LIN {X 0,Y 325.669,Z 599.39,A -85,B 0,C 180,E1 -14857.439,E2 -14857.439} C_VEL
LIN {X 0,Y 325.677,Z 594.579,A -85,B 0,C 180,E1 -14859.314,E2 -14859.314} C_VEL
LIN {X 0,Y 326.028,Z 587.351,A -85,B 0,C 180,E1 -14861.501,E2 -14861.501} C_VEL
LIN {X 0,Y 326.643,Z 579.568,A -85,B 0,C 180,E1 -14863.373,E2 -14863.373} C_VEL
LIN {X 0,Y 327.397,Z 571.651,A -85,B 0,C 180,E1 -14864.927,E2 -14864.927} C_VEL
LIN {X 0,Y 328.601,Z 562.062,A -85,B 0,C 180,E1 -14866.462,E2 -14866.462} C_VEL
LIN {X 0,Y 329.683,Z 551.406,A -85,B 0,C 180,E1 -14867.845,E2 -14867.845} C_VEL
LIN {X 0,Y 329.651,Z 539.37,A -85,B 0,C 180,E1 -14869.134,E2 -14869.134} C_VEL
LIN {X 0,Y 329.259,Z 526.597,A -85,B 0,C 180,E1 -14870.206,E2 -14870.206} C_VEL
LIN {X 0,Y 328.339,Z 513.613,A -85,B 0,C 180,E1 -14871.05,E2 -14871.05} C_VEL
LIN {X 0,Y 326.76,Z 500.315,A -85,B 0,C 180,E1 -14871.695,E2 -14871.695} C_VEL
LIN {X 0,Y 326.159,Z 495.999,A -85,B 0,C 180,E1 -14871.874,E2 -14871.874} C_VEL
LIN {X 0,Y 327.015,Z 484.007,A -85,B 0,C 180,E1 -14876.14,E2 -14876.14} C_VEL
LIN {X 0,Y 328.094,Z 472.597,A -85,B 0,C 180,E1 -14880.224,E2 -14880.224} C_VEL
LIN {X 0,Y 329.193,Z 462.925,A -85,B 0,C 180,E1 -14883.716,E2 -14883.716} C_VEL
LIN {X 0,Y 330.448,Z 453.169,A -85,B 0,C 180,E1 -14887.311,E2 -14887.311} C_VEL
LIN {X 0,Y 330.5,Z 451.076,A -85,B 0,C 180,E1 -14888.113,E2 -14888.113} C_VEL
LIN {X 0,Y 328.983,Z 442.588,A -85,B 0,C 180,E1 -14891.609,E2 -14891.609} C_VEL
LIN {X 0,Y 327.405,Z 434.615,A -85,B 0,C 180,E1 -14895.102,E2 -14895.102} C_VEL
LIN {X 0,Y 326.602,Z 430.809,A -85,B 0,C 180,E1 -14896.887,E2 -14896.887} C_VEL
LIN {X 0,Y 326.612,Z 430.8,A -85,B 0,C 180,E1 -14900.772,E2 -14900.772} C_VEL
LIN {X 0,Y 326.614,Z 430.802,A -85,B 0,C 180,E1 -14904.481,E2 -14904.481} C_VEL
LIN {X 0,Y 326.61,Z 430.799,A -85,B 0,C 180,E1 -14907.456,E2 -14907.456} C_VEL
LIN {X 0,Y 326.648,Z 430.798,A -85,B 0,C 180,E1 -14910.34,E2 -14910.34} C_VEL
LIN {X 0,Y 326.69,Z 430.791,A -85,B 0,C 180,E1 -14914.516,E2 -14914.516} C_VEL
LIN {X 0,Y 326.649,Z 430.796,A -85,B 0,C 180,E1 -14918.546,E2 -14918.546} C_VEL
LIN {X 0,Y 326.745,Z 430.782,A -85,B 0,C 180,E1 -14921.178,E2 -14921.178} C_VEL
LIN {X 0,Y 326.764,Z 430.78,A -85,B 0,C 180,E1 -14925.433,E2 -14925.433} C_VEL
LIN {X 0,Y 326.774,Z 430.778,A -85,B 0,C 180,E1 -14928.839,E2 -14928.839} C_VEL
LIN {X 0,Y 326.945,Z 430.758,A -85,B 0,C 180,E1 -14932.59,E2 -14932.59} C_VEL
LIN {X 0,Y 326.986,Z 430.755,A -85,B 0,C 180,E1 -14933.831,E2 -14933.831} C_VEL
LIN {X 0,Y 327.05,Z 430.745,A -85,B 0,C 180,E1 -14937.537,E2 -14937.537} C_VEL
LIN {X 0,Y 327.218,Z 430.728,A -85,B 0,C 180,E1 -14940,E2 -14940} C_VEL
LIN {X 0,Y 327.047,Z 430.745,A -85,B 0,C 180,E1 -14942.463,E2 -14942.463} C_VEL
LIN {X 0,Y 326.972,Z 430.752,A -85,B 0,C 180,E1 -14946.678,E2 -14946.678} C_VEL
LIN {X 0,Y 326.815,Z 430.777,A -85,B 0,C 180,E1 -14949.906,E2 -14949.906} C_VEL
LIN {X 0,Y 326.76,Z 430.78,A -85,B 0,C 180,E1 -14953.686,E2 -14953.686} C_VEL
LIN {X 0,Y 326.701,Z 430.788,A -85,B 0,C 180,E1 -14957.528,E2 -14957.528} C_VEL
LIN {X 0,Y 326.666,Z 430.79,A -85,B 0,C 180,E1 -14960.135,E2 -14960.135} C_VEL
LIN {X 0,Y 326.653,Z 430.794,A -85,B 0,C 180,E1 -14964.129,E2 -14964.129} C_VEL
LIN {X 0,Y 326.684,Z 430.788,A -85,B 0,C 180,E1 -14966.858,E2 -14966.858} C_VEL
LIN {X 0,Y 326.635,Z 430.794,A -85,B 0,C 180,E1 -14970.61,E2 -14970.61} C_VEL
LIN {X 0,Y 326.609,Z 430.8,A -85,B 0,C 180,E1 -14974.02,E2 -14974.02} C_VEL
LIN {X 0,Y 326.629,Z 430.796,A -85,B 0,C 180,E1 -14977.239,E2 -14977.239} C_VEL
LIN {X 0,Y 326.579,Z 430.801,A -85,B 0,C 180,E1 -14981.132,E2 -14981.132} C_VEL
LIN {X 0,Y 326.53,Z 430.807,A -85,B 0,C 180,E1 -14984.743,E2 -14984.743} C_VEL
LIN {X 0,Y 326.578,Z 430.803,A -85,B 0,C 180,E1 -14988.155,E2 -14988.155} C_VEL
LIN {X 0,Y 326.626,Z 430.797,A -85,B 0,C 180,E1 -14991.392,E2 -14991.392} C_VEL
LIN {X 0,Y 326.622,Z 430.795,A -85,B 0,C 180,E1 -14994.852,E2 -14994.852} C_VEL
LIN {X 0,Y 326.618,Z 430.799,A -85,B 0,C 180,E1 -14997.457,E2 -14997.457} C_VEL
LIN {X 0,Y 326.664,Z 430.79,A -85,B 0,C 180,E1 -15000.342,E2 -15000.342} C_VEL
LIN {X 0,Y 326.688,Z 430.789,A -85,B 0,C 180,E1 -15003.143,E2 -15003.143} C_VEL
LIN {X 0,Y 326.655,Z 430.797,A -85,B 0,C 180,E1 -15005.872,E2 -15005.872} C_VEL
LIN {X 0,Y 326.671,Z 430.795,A -85,B 0,C 180,E1 -15009.866,E2 -15009.866} C_VEL
LIN {X 0,Y 326.767,Z 430.78,A -85,B 0,C 180,E1 -15012.234,E2 -15012.234} C_VEL
LIN {X 0,Y 330.786,Z 443.096,A -85,B 0,C 180,E1 -15013.451,E2 -15013.451} C_VEL
LIN {X 0,Y 333.898,Z 454.069,A -85,B 0,C 180,E1 -15014.746,E2 -15014.746} C_VEL
LIN {X 0,Y 333.148,Z 464.325,A -85,B 0,C 180,E1 -15015.961,E2 -15015.961} C_VEL
LIN {X 0,Y 331.99,Z 474.107,A -85,B 0,C 180,E1 -15017.371,E2 -15017.371} C_VEL
LIN {X 0,Y 330.794,Z 483.132,A -85,B 0,C 180,E1 -15018.977,E2 -15018.977} C_VEL
LIN {X 0,Y 329.724,Z 491.285,A -85,B 0,C 180,E1 -15020.801,E2 -15020.801} C_VEL
LIN {X 0,Y 328.764,Z 497.856,A -85,B 0,C 180,E1 -15022.631,E2 -15022.631} C_VEL
LIN {X 0,Y 328.229,Z 503.065,A -85,B 0,C 180,E1 -15024.471,E2 -15024.471} C_VEL
LIN {X 0,Y 327.548,Z 507.179,A -85,B 0,C 180,E1 -15026.31,E2 -15026.31} C_VEL
LIN {X 0,Y 327.213,Z 509.362,A -85,B 0,C 180,E1 -15027.538,E2 -15027.538} C_VEL
LIN {X 0,Y 326.991,Z 511.075,A -85,B 0,C 180,E1 -15028.769,E2 -15028.769} C_VEL
LIN {X 0,Y 326.874,Z 513.281,A -85,B 0,C 180,E1 -15031.232,E2 -15031.232} C_VEL
LIN {X 0,Y 326.764,Z 513.841,A -85,B 0,C 180,E1 -15032.466,E2 -15032.466} C_VEL
LIN {X 0,Y 326.652,Z 513.995,A -85,B 0,C 180,E1 -15033.701,E2 -15033.701} C_VEL
LIN {X 0,Y 327.059,Z 513.1,A -85,B 0,C 180,E1 -15036.168,E2 -15036.168} C_VEL
LIN {X 0,Y 327.451,Z 512.077,A -85,B 0,C 180,E1 -15037.399,E2 -15037.399} C_VEL
LIN {X 0,Y 328.031,Z 508.988,A -85,B 0,C 180,E1 -15039.752,E2 -15039.752} C_VEL
LIN {X 0,Y 328.83,Z 505.182,A -85,B 0,C 180,E1 -15041.715,E2 -15041.715} C_VEL
LIN {X 0,Y 329.619,Z 500.482,A -85,B 0,C 180,E1 -15043.565,E2 -15043.565} C_VEL
LIN {X 0,Y 330.597,Z 494.526,A -85,B 0,C 180,E1 -15045.411,E2 -15045.411} C_VEL
LIN {X 0,Y 331.772,Z 487.085,A -85,B 0,C 180,E1 -15047.252,E2 -15047.252} C_VEL
LIN {X 0,Y 333.026,Z 479.414,A -85,B 0,C 180,E1 -15048.774,E2 -15048.774} C_VEL
LIN {X 0,Y 334.289,Z 468.983,A -85,B 0,C 180,E1 -15050.458,E2 -15050.458} C_VEL
LIN {X 0,Y 335.431,Z 459.35,A -85,B 0,C 180,E1 -15051.7,E2 -15051.7} C_VEL
LIN {X 0,Y 335.445,Z 457.058,A -85,B 0,C 180,E1 -15051.978,E2 -15051.978} C_VEL
LIN {X 0,Y 332.16,Z 446.15,A -85,B 0,C 180,E1 -15053.401,E2 -15053.401} C_VEL
LIN {X 0,Y 328.166,Z 435.083,A -85,B 0,C 180,E1 -15054.651,E2 -15054.651} C_VEL
LIN {X 0,Y 326.687,Z 430.788,A -85,B 0,C 180,E1 -15055.101,E2 -15055.101} C_VEL
LIN {X 0,Y 326.66,Z 430.797,A -85,B 0,C 180,E1 -15058.251,E2 -15058.251} C_VEL
LIN {X 0,Y 326.598,Z 430.801,A -85,B 0,C 180,E1 -15061.095,E2 -15061.095} C_VEL
LIN {X 0,Y 326.612,Z 430.803,A -85,B 0,C 180,E1 -15064.019,E2 -15064.019} C_VEL
LIN {X 0,Y 326.631,Z 430.796,A -85,B 0,C 180,E1 -15067.239,E2 -15067.239} C_VEL
LIN {X 0,Y 326.581,Z 430.802,A -85,B 0,C 180,E1 -15071.131,E2 -15071.131} C_VEL
LIN {X 0,Y 326.532,Z 430.808,A -85,B 0,C 180,E1 -15074.743,E2 -15074.743} C_VEL
LIN {X 0,Y 326.58,Z 430.806,A -85,B 0,C 180,E1 -15078.154,E2 -15078.154} C_VEL
LIN {X 0,Y 326.627,Z 430.796,A -85,B 0,C 180,E1 -15081.391,E2 -15081.391} C_VEL
LIN {X 0,Y 326.623,Z 430.796,A -85,B 0,C 180,E1 -15084.851,E2 -15084.851} C_VEL
LIN {X 0,Y 326.614,Z 430.799,A -85,B 0,C 180,E1 -15087.456,E2 -15087.456} C_VEL
LIN {X 0,Y 326.664,Z 430.793,A -85,B 0,C 180,E1 -15090.341,E2 -15090.341} C_VEL
LIN {X 0,Y 326.694,Z 430.788,A -85,B 0,C 180,E1 -15094.516,E2 -15094.516} C_VEL
LIN {X 0,Y 326.655,Z 430.792,A -85,B 0,C 180,E1 -15095.197,E2 -15095.197} C_VEL
LIN {X 0,Y 325.957,Z 430.883,A -85,B 0,C 180,E1 -15096.225,E2 -15096.225} C_VEL
LIN {X 0,Y 323.068,Z 431.244,A -85,B 0,C 180,E1 -15097.898,E2 -15097.898} C_VEL
LIN {X 0,Y 320.677,Z 431.538,A -85,B 0,C 180,E1 -15099.254,E2 -15099.254} C_VEL
LIN {X 0,Y 319.714,Z 431.658,A -85,B 0,C 180,E1 -15100.304,E2 -15100.304} C_VEL
LIN {X 0,Y 319.668,Z 431.662,A -85,B 0,C 180,E1 -15100.659,E2 -15100.659} C_VEL
LIN {X 0,Y 319.742,Z 431.745,A -85,B 0,C 180,E1 -15102.367,E2 -15102.367} C_VEL
LIN {X 0,Y 322.789,Z 444.313,A -85,B 0,C 180,E1 -15103.558,E2 -15103.558} C_VEL
LIN {X 0,Y 323.928,Z 449.817,A -85,B 0,C 180,E1 -15104.161,E2 -15104.161} C_VEL
LIN {X 0,Y 323.077,Z 461.417,A -85,B 0,C 180,E1 -15105.513,E2 -15105.513} C_VEL
LIN {X 0,Y 322.358,Z 472.344,A -85,B 0,C 180,E1 -15107.087,E2 -15107.087} C_VEL
LIN {X 0,Y 321.437,Z 483.009,A -85,B 0,C 180,E1 -15108.97,E2 -15108.97} C_VEL
LIN {X 0,Y 320.873,Z 491.396,A -85,B 0,C 180,E1 -15110.814,E2 -15110.814} C_VEL
LIN {X 0,Y 320.306,Z 498.633,A -85,B 0,C 180,E1 -15112.752,E2 -15112.752} C_VEL
LIN {X 0,Y 319.786,Z 505.159,A -85,B 0,C 180,E1 -15114.956,E2 -15114.956} C_VEL
LIN {X 0,Y 319.604,Z 509.482,A -85,B 0,C 180,E1 -15116.848,E2 -15116.848} C_VEL
LIN {X 0,Y 319.665,Z 512.75,A -85,B 0,C 180,E1 -15118.74,E2 -15118.74} C_VEL
LIN {X 0,Y 319.823,Z 514.387,A -85,B 0,C 180,E1 -15120,E2 -15120} C_VEL
LIN {X 0,Y 319.913,Z 515.65,A -85,B 0,C 180,E1 -15121.259,E2 -15121.259} C_VEL
LIN {X 0,Y 320.345,Z 516.87,A -85,B 0,C 180,E1 -15123.774,E2 -15123.774} C_VEL
LIN {X 0,Y 320.674,Z 516.901,A -85,B 0,C 180,E1 -15125.029,E2 -15125.029} C_VEL
LIN {X 0,Y 321.105,Z 516.495,A -85,B 0,C 180,E1 -15126.283,E2 -15126.283} C_VEL
LIN {X 0,Y 322.298,Z 514.492,A -85,B 0,C 180,E1 -15128.78,E2 -15128.78} C_VEL
LIN {X 0,Y 323.367,Z 511.902,A -85,B 0,C 180,E1 -15130.646,E2 -15130.646} C_VEL
LIN {X 0,Y 324.733,Z 508.273,A -85,B 0,C 180,E1 -15132.499,E2 -15132.499} C_VEL
LIN {X 0,Y 326.445,Z 502.775,A -85,B 0,C 180,E1 -15134.621,E2 -15134.621} C_VEL
LIN {X 0,Y 328.227,Z 496.576,A -85,B 0,C 180,E1 -15136.482,E2 -15136.482} C_VEL
LIN {X 0,Y 330.281,Z 488.982,A -85,B 0,C 180,E1 -15138.292,E2 -15138.292} C_VEL
LIN {X 0,Y 332.466,Z 479.622,A -85,B 0,C 180,E1 -15140.091,E2 -15140.091} C_VEL
LIN {X 0,Y 334.516,Z 470.377,A -85,B 0,C 180,E1 -15141.521,E2 -15141.521} C_VEL
LIN {X 0,Y 335.117,Z 467.023,A -85,B 0,C 180,E1 -15141.982,E2 -15141.982} C_VEL
LIN {X 0,Y 332.872,Z 458.578,A -85,B 0,C 180,E1 -15143.65,E2 -15143.65} C_VEL
LIN {X 0,Y 329.131,Z 449.041,A -85,B 0,C 180,E1 -15145.596,E2 -15145.596} C_VEL
LIN {X 0,Y 324.805,Z 440.543,A -85,B 0,C 180,E1 -15147.483,E2 -15147.483} C_VEL
LIN {X 0,Y 322.807,Z 437.235,A -85,B 0,C 180,E1 -15148.282,E2 -15148.282} C_VEL
LIN {X 0,Y 320.236,Z 433.853,A -85,B 0,C 180,E1 -15149.259,E2 -15149.259} C_VEL
LIN {X 0,Y 319.626,Z 431.669,A -85,B 0,C 180,E1 -15149.652,E2 -15149.652} C_VEL
LIN {X 0,Y 319.579,Z 431.674,A -85,B 0,C 180,E1 -15153.352,E2 -15153.352} C_VEL
LIN {X 0,Y 319.561,Z 431.681,A -85,B 0,C 180,E1 -15156.427,E2 -15156.427} C_VEL
LIN {X 0,Y 319.565,Z 431.681,A -85,B 0,C 180,E1 -15160.449,E2 -15160.449} C_VEL
LIN {X 0,Y 319.588,Z 431.813,A -85,B 0,C 180,E1 -15160.861,E2 -15160.861} C_VEL
LIN {X 0,Y 321.083,Z 439.049,A -85,B 0,C 180,E1 -15164.461,E2 -15164.461} C_VEL
LIN {X 0,Y 322.551,Z 446.207,A -85,B 0,C 180,E1 -15167.801,E2 -15167.801} C_VEL
LIN {X 0,Y 323.926,Z 453.523,A -85,B 0,C 180,E1 -15171.009,E2 -15171.009} C_VEL
LIN {X 0,Y 324.151,Z 455.88,A -85,B 0,C 180,E1 -15171.991,E2 -15171.991} C_VEL
LIN {X 0,Y 322.624,Z 465.941,A -85,B 0,C 180,E1 -15175.872,E2 -15175.872} C_VEL
LIN {X 0,Y 321.265,Z 476.33,A -85,B 0,C 180,E1 -15179.791,E2 -15179.791} C_VEL
LIN {X 0,Y 320.595,Z 482.587,A -85,B 0,C 180,E1 -15182.058,E2 -15182.058} C_VEL
LIN {X 0,Y 321.374,Z 486.979,A -85,B 0,C 180,E1 -15182.529,E2 -15182.529} C_VEL
LIN {X 0,Y 323.338,Z 495.524,A -85,B 0,C 180,E1 -15183.548,E2 -15183.548} C_VEL
LIN {X 0,Y 325.59,Z 511.177,A -85,B 0,C 180,E1 -15185.304,E2 -15185.304} C_VEL
LIN {X 0,Y 326.507,Z 524.117,A -85,B 0,C 180,E1 -15186.797,E2 -15186.797} C_VEL
LIN {X 0,Y 326.004,Z 535.939,A -85,B 0,C 180,E1 -15188.199,E2 -15188.199} C_VEL
LIN {X 0,Y 324.904,Z 548.75,A -85,B 0,C 180,E1 -15189.916,E2 -15189.916} C_VEL
LIN {X 0,Y 323.91,Z 557.8,A -85,B 0,C 180,E1 -15191.334,E2 -15191.334} C_VEL
LIN {X 0,Y 321.843,Z 568.154,A -85,B 0,C 180,E1 -15193.181,E2 -15193.181} C_VEL
LIN {X 0,Y 319.919,Z 581.019,A -85,B 0,C 180,E1 -15196.016,E2 -15196.016} C_VEL
LIN {X 0,Y 319.057,Z 588.233,A -85,B 0,C 180,E1 -15197.921,E2 -15197.921} C_VEL
LIN {X 0,Y 318.563,Z 594.058,A -85,B 0,C 180,E1 -15199.834,E2 -15199.834} C_VEL
LIN {X 0,Y 318.512,Z 598.707,A -85,B 0,C 180,E1 -15201.754,E2 -15201.754} C_VEL
LIN {X 0,Y 318.634,Z 602.266,A -85,B 0,C 180,E1 -15203.668,E2 -15203.668} C_VEL
LIN {X 0,Y 318.818,Z 604.062,A -85,B 0,C 180,E1 -15204.941,E2 -15204.941} C_VEL
LIN {X 0,Y 318.996,Z 605.438,A -85,B 0,C 180,E1 -15206.21,E2 -15206.21} C_VEL
LIN {X 0,Y 319.08,Z 606.386,A -85,B 0,C 180,E1 -15207.475,E2 -15207.475} C_VEL
LIN {X 0,Y 319.469,Z 606.925,A -85,B 0,C 180,E1 -15208.739,E2 -15208.739} C_VEL
LIN {X 0,Y 319.619,Z 607.015,A -85,B 0,C 180,E1 -15210,E2 -15210} C_VEL
LIN {X 0,Y 319.487,Z 606.66,A -85,B 0,C 180,E1 -15211.26,E2 -15211.26} C_VEL
LIN {X 0,Y 319.132,Z 605.866,A -85,B 0,C 180,E1 -15212.524,E2 -15212.524} C_VEL
LIN {X 0,Y 319.046,Z 604.651,A -85,B 0,C 180,E1 -15213.789,E2 -15213.789} C_VEL
LIN {X 0,Y 318.806,Z 602.006,A -85,B 0,C 180,E1 -15215.693,E2 -15215.693} C_VEL
LIN {X 0,Y 318.604,Z 598.302,A -85,B 0,C 180,E1 -15217.605,E2 -15217.605} C_VEL
LIN {X 0,Y 318.615,Z 593.468,A -85,B 0,C 180,E1 -15219.522,E2 -15219.522} C_VEL
LIN {X 0,Y 319.018,Z 586.22,A -85,B 0,C 180,E1 -15221.758,E2 -15221.758} C_VEL
LIN {X 0,Y 319.692,Z 578.418,A -85,B 0,C 180,E1 -15223.669,E2 -15223.669} C_VEL
LIN {X 0,Y 320.297,Z 571.806,A -85,B 0,C 180,E1 -15225.005,E2 -15225.005} C_VEL
LIN {X 0,Y 321.504,Z 562.93,A -85,B 0,C 180,E1 -15226.509,E2 -15226.509} C_VEL
LIN {X 0,Y 322.676,Z 552.778,A -85,B 0,C 180,E1 -15227.917,E2 -15227.917} C_VEL
LIN {X 0,Y 322.689,Z 541.461,A -85,B 0,C 180,E1 -15229.215,E2 -15229.215} C_VEL
LIN {X 0,Y 322.447,Z 528.376,A -85,B 0,C 180,E1 -15230.41,E2 -15230.41} C_VEL
LIN {X 0,Y 321.673,Z 515.529,A -85,B 0,C 180,E1 -15231.319,E2 -15231.319} C_VEL
LIN {X 0,Y 320.175,Z 502.104,A -85,B 0,C 180,E1 -15232.032,E2 -15232.032} C_VEL
LIN {X 0,Y 319.167,Z 494.914,A -85,B 0,C 180,E1 -15232.357,E2 -15232.357} C_VEL
LIN {X 0,Y 320.089,Z 482.916,A -85,B 0,C 180,E1 -15236.75,E2 -15236.75} C_VEL
LIN {X 0,Y 321.44,Z 470.016,A -85,B 0,C 180,E1 -15241.493,E2 -15241.493} C_VEL
LIN {X 0,Y 322.624,Z 459.929,A -85,B 0,C 180,E1 -15245.259,E2 -15245.259} C_VEL
LIN {X 0,Y 323.456,Z 454.085,A -85,B 0,C 180,E1 -15247.472,E2 -15247.472} C_VEL
LIN {X 0,Y 323.155,Z 450.05,A -85,B 0,C 180,E1 -15249.101,E2 -15249.101} C_VEL
LIN {X 0,Y 321.624,Z 441.786,A -85,B 0,C 180,E1 -15252.641,E2 -15252.641} C_VEL
LIN {X 0,Y 319.907,Z 433.467,A -85,B 0,C 180,E1 -15256.466,E2 -15256.466} C_VEL
LIN {X 0,Y 319.535,Z 431.689,A -85,B 0,C 180,E1 -15257.39,E2 -15257.39} C_VEL
LIN {X 0,Y 319.548,Z 431.683,A -85,B 0,C 180,E1 -15260.371,E2 -15260.371} C_VEL
LIN {X 0,Y 319.56,Z 431.678,A -85,B 0,C 180,E1 -15263.573,E2 -15263.573} C_VEL
LIN {X 0,Y 319.577,Z 431.677,A -85,B 0,C 180,E1 -15266.686,E2 -15266.686} C_VEL
LIN {X 0,Y 319.585,Z 431.675,A -85,B 0,C 180,E1 -15269.616,E2 -15269.616} C_VEL
LIN {X 0,Y 319.606,Z 431.673,A -85,B 0,C 180,E1 -15272.498,E2 -15272.498} C_VEL
LIN {X 0,Y 319.605,Z 431.671,A -85,B 0,C 180,E1 -15275.304,E2 -15275.304} C_VEL
LIN {X 0,Y 319.598,Z 431.677,A -85,B 0,C 180,E1 -15278.048,E2 -15278.048} C_VEL
LIN {X 0,Y 319.69,Z 431.661,A -85,B 0,C 180,E1 -15280.962,E2 -15280.962} C_VEL
LIN {X 0,Y 319.731,Z 431.656,A -85,B 0,C 180,E1 -15285.276,E2 -15285.276} C_VEL
LIN {X 0,Y 319.754,Z 431.656,A -85,B 0,C 180,E1 -15289.873,E2 -15289.873} C_VEL
LIN {X 0,Y 319.939,Z 431.631,A -85,B 0,C 180,E1 -15293.694,E2 -15293.694} C_VEL
LIN {X 0,Y 319.994,Z 431.623,A -85,B 0,C 180,E1 -15297.483,E2 -15297.483} C_VEL
LIN {X 0,Y 320.17,Z 431.606,A -85,B 0,C 180,E1 -15300,E2 -15300} C_VEL
LIN {X 0,Y 319.991,Z 431.624,A -85,B 0,C 180,E1 -15302.518,E2 -15302.518} C_VEL
LIN {X 0,Y 319.932,Z 431.629,A -85,B 0,C 180,E1 -15306.669,E2 -15306.669} C_VEL
LIN {X 0,Y 319.759,Z 431.655,A -85,B 0,C 180,E1 -15310.127,E2 -15310.127} C_VEL
LIN {X 0,Y 319.732,Z 431.654,A -85,B 0,C 180,E1 -15314.725,E2 -15314.725} C_VEL
LIN {X 0,Y 319.69,Z 431.658,A -85,B 0,C 180,E1 -15319.038,E2 -15319.038} C_VEL
LIN {X 0,Y 319.571,Z 431.669,A -85,B 0,C 180,E1 -15323.32,E2 -15323.32} C_VEL
LIN {X 0,Y 319.635,Z 431.67,A -85,B 0,C 180,E1 -15326.088,E2 -15326.088} C_VEL
LIN {X 0,Y 319.581,Z 431.673,A -85,B 0,C 180,E1 -15328.935,E2 -15328.935} C_VEL
LIN {X 0,Y 319.533,Z 431.68,A -85,B 0,C 180,E1 -15331.862,E2 -15331.862} C_VEL
LIN {X 0,Y 319.581,Z 431.673,A -85,B 0,C 180,E1 -15335.543,E2 -15335.543} C_VEL
LIN {X 0,Y 319.575,Z 431.678,A -85,B 0,C 180,E1 -15338.008,E2 -15338.008} C_VEL
LIN {X 0,Y 319.527,Z 431.683,A -85,B 0,C 180,E1 -15341.597,E2 -15341.597} C_VEL
LIN {X 0,Y 319.491,Z 431.684,A -85,B 0,C 180,E1 -15345.258,E2 -15345.258} C_VEL
LIN {X 0,Y 319.53,Z 431.678,A -85,B 0,C 180,E1 -15348.712,E2 -15348.712} C_VEL
LIN {X 0,Y 319.579,Z 431.674,A -85,B 0,C 180,E1 -15352.344,E2 -15352.344} C_VEL
LIN {X 0,Y 319.563,Z 431.675,A -85,B 0,C 180,E1 -15355.124,E2 -15355.124} C_VEL
LIN {X 0,Y 319.577,Z 431.674,A -85,B 0,C 180,E1 -15359.057,E2 -15359.057} C_VEL
LIN {X 0,Y 319.62,Z 431.669,A -85,B 0,C 180,E1 -15362.499,E2 -15362.499} C_VEL
LIN {X 0,Y 319.608,Z 431.672,A -85,B 0,C 180,E1 -15365.304,E2 -15365.304} C_VEL
LIN {X 0,Y 319.601,Z 431.675,A -85,B 0,C 180,E1 -15368.048,E2 -15368.048} C_VEL
LIN {X 0,Y 319.744,Z 431.655,A -85,B 0,C 180,E1 -15371.782,E2 -15371.782} C_VEL
LIN {X 0,Y 323.953,Z 444.512,A -85,B 0,C 180,E1 -15373.084,E2 -15373.084} C_VEL
LIN {X 0,Y 327.063,Z 455.441,A -85,B 0,C 180,E1 -15374.419,E2 -15374.419} C_VEL
LIN {X 0,Y 326.814,Z 460.778,A -85,B 0,C 180,E1 -15375.046,E2 -15375.046} C_VEL
LIN {X 0,Y 325.617,Z 471.249,A -85,B 0,C 180,E1 -15376.451,E2 -15376.451} C_VEL
LIN {X 0,Y 324.617,Z 479.482,A -85,B 0,C 180,E1 -15377.814,E2 -15377.814} C_VEL
LIN {X 0,Y 323.586,Z 487.223,A -85,B 0,C 180,E1 -15379.362,E2 -15379.362} C_VEL
LIN {X 0,Y 322.425,Z 494.811,A -85,B 0,C 180,E1 -15381.224,E2 -15381.224} C_VEL
LIN {X 0,Y 321.694,Z 500.842,A -85,B 0,C 180,E1 -15383.099,E2 -15383.099} C_VEL
LIN {X 0,Y 320.985,Z 505.658,A -85,B 0,C 180,E1 -15384.976,E2 -15384.976} C_VEL
LIN {X 0,Y 320.398,Z 509.39,A -85,B 0,C 180,E1 -15386.857,E2 -15386.857} C_VEL
LIN {X 0,Y 319.97,Z 512.13,A -85,B 0,C 180,E1 -15388.742,E2 -15388.742} C_VEL
LIN {X 0,Y 319.852,Z 514.316,A -85,B 0,C 180,E1 -15391.259,E2 -15391.259} C_VEL
LIN {X 0,Y 319.74,Z 514.865,A -85,B 0,C 180,E1 -15392.52,E2 -15392.52} C_VEL
LIN {X 0,Y 319.631,Z 515.003,A -85,B 0,C 180,E1 -15393.782,E2 -15393.782} C_VEL
LIN {X 0,Y 320.067,Z 514.088,A -85,B 0,C 180,E1 -15396.303,E2 -15396.303} C_VEL
LIN {X 0,Y 320.477,Z 513.053,A -85,B 0,C 180,E1 -15397.561,E2 -15397.561} C_VEL
LIN {X 0,Y 321.106,Z 509.937,A -85,B 0,C 180,E1 -15399.964,E2 -15399.964} C_VEL
LIN {X 0,Y 321.946,Z 506.107,A -85,B 0,C 180,E1 -15401.969,E2 -15401.969} C_VEL
LIN {X 0,Y 322.76,Z 501.387,A -85,B 0,C 180,E1 -15403.859,E2 -15403.859} C_VEL
LIN {X 0,Y 323.805,Z 495.404,A -85,B 0,C 180,E1 -15405.742,E2 -15405.742} C_VEL
LIN {X 0,Y 325.048,Z 487.925,A -85,B 0,C 180,E1 -15407.62,E2 -15407.62} C_VEL
LIN {X 0,Y 326.602,Z 478.461,A -85,B 0,C 180,E1 -15409.484,E2 -15409.484} C_VEL
LIN {X 0,Y 327.835,Z 468.682,A -85,B 0,C 180,E1 -15411.044,E2 -15411.044} C_VEL
LIN {X 0,Y 328.936,Z 459.565,A -85,B 0,C 180,E1 -15412.213,E2 -15412.213} C_VEL
LIN {X 0,Y 326.001,Z 449.452,A -85,B 0,C 180,E1 -15413.604,E2 -15413.604} C_VEL
LIN {X 0,Y 322.562,Z 439.477,A -85,B 0,C 180,E1 -15414.802,E2 -15414.802} C_VEL
LIN {X 0,Y 319.639,Z 431.667,A -85,B 0,C 180,E1 -15415.646,E2 -15415.646} C_VEL
LIN {X 0,Y 319.593,Z 431.674,A -85,B 0,C 180,E1 -15418.934,E2 -15418.934} C_VEL
LIN {X 0,Y 319.537,Z 431.683,A -85,B 0,C 180,E1 -15421.862,E2 -15421.862} C_VEL
LIN {X 0,Y 319.584,Z 431.674,A -85,B 0,C 180,E1 -15425.543,E2 -15425.543} C_VEL
LIN {X 0,Y 319.577,Z 431.679,A -85,B 0,C 180,E1 -15428.008,E2 -15428.008} C_VEL
LIN {X 0,Y 319.529,Z 431.682,A -85,B 0,C 180,E1 -15431.597,E2 -15431.597} C_VEL
LIN {X 0,Y 319.492,Z 431.685,A -85,B 0,C 180,E1 -15435.257,E2 -15435.257} C_VEL
LIN {X 0,Y 319.532,Z 431.68,A -85,B 0,C 180,E1 -15438.712,E2 -15438.712} C_VEL
LIN {X 0,Y 319.581,Z 431.676,A -85,B 0,C 180,E1 -15442.344,E2 -15442.344} C_VEL
LIN {X 0,Y 319.564,Z 431.675,A -85,B 0,C 180,E1 -15445.123,E2 -15445.123} C_VEL
LIN {X 0,Y 319.574,Z 431.674,A -85,B 0,C 180,E1 -15449.058,E2 -15449.058} C_VEL
LIN {X 0,Y 319.612,Z 431.67,A -85,B 0,C 180,E1 -15452.498,E2 -15452.498} C_VEL
LIN {X 0,Y 319.607,Z 431.671,A -85,B 0,C 180,E1 -15455.304,E2 -15455.304} C_VEL
LIN {X 0,Y 319.607,Z 431.672,A -85,B 0,C 180,E1 -15459.4,E2 -15459.4} C_VEL
LIN {X 0,Y 319.668,Z 431.662,A -85,B 0,C 180,E1 -15460.659,E2 -15460.659} C_VEL
LIN {X 0,Y 319.605,Z 432.418,A -85,B 0,C 180,E1 -15461.315,E2 -15461.315} C_VEL
LIN {X 0,Y 319.347,Z 434.282,A -85,B 0,C 180,E1 -15461.905,E2 -15461.905} C_VEL
LIN {X 0,Y 318.737,Z 438.373,A -85,B 0,C 180,E1 -15462.654,E2 -15462.654} C_VEL
LIN {X 0,Y 317.424,Z 447.32,A -85,B 0,C 180,E1 -15463.66,E2 -15463.66} C_VEL
LIN {X 0,Y 316.584,Z 454.78,A -85,B 0,C 180,E1 -15464.445,E2 -15464.445} C_VEL
LIN {X 0,Y 315.767,Z 466.772,A -85,B 0,C 180,E1 -15465.993,E2 -15465.993} C_VEL
LIN {X 0,Y 315.036,Z 476.021,A -85,B 0,C 180,E1 -15467.437,E2 -15467.437} C_VEL
LIN {X 0,Y 314.26,Z 486.148,A -85,B 0,C 180,E1 -15469.368,E2 -15469.368} C_VEL
LIN {X 0,Y 313.6,Z 494.412,A -85,B 0,C 180,E1 -15471.299,E2 -15471.299} C_VEL
LIN {X 0,Y 313.031,Z 502.069,A -85,B 0,C 180,E1 -15473.554,E2 -15473.554} C_VEL
LIN {X 0,Y 312.709,Z 507.3,A -85,B 0,C 180,E1 -15475.488,E2 -15475.488} C_VEL
LIN {X 0,Y 312.568,Z 510.173,A -85,B 0,C 180,E1 -15476.777,E2 -15476.777} C_VEL
LIN {X 0,Y 312.639,Z 513.581,A -85,B 0,C 180,E1 -15478.712,E2 -15478.712} C_VEL
LIN {X 0,Y 312.799,Z 515.288,A -85,B 0,C 180,E1 -15480,E2 -15480} C_VEL
LIN {X 0,Y 312.894,Z 516.625,A -85,B 0,C 180,E1 -15481.287,E2 -15481.287} C_VEL
LIN {X 0,Y 313.083,Z 517.548,A -85,B 0,C 180,E1 -15482.573,E2 -15482.573} C_VEL
LIN {X 0,Y 313.708,Z 518.135,A -85,B 0,C 180,E1 -15485.141,E2 -15485.141} C_VEL
LIN {X 0,Y 314.179,Z 517.857,A -85,B 0,C 180,E1 -15486.422,E2 -15486.422} C_VEL
LIN {X 0,Y 314.741,Z 517.134,A -85,B 0,C 180,E1 -15487.699,E2 -15487.699} C_VEL
LIN {X 0,Y 316.189,Z 514.487,A -85,B 0,C 180,E1 -15490.243,E2 -15490.243} C_VEL
LIN {X 0,Y 317.513,Z 511.395,A -85,B 0,C 180,E1 -15492.138,E2 -15492.138} C_VEL
LIN {X 0,Y 319.048,Z 507.272,A -85,B 0,C 180,E1 -15494.023,E2 -15494.023} C_VEL
LIN {X 0,Y 321.137,Z 500.945,A -85,B 0,C 180,E1 -15496.202,E2 -15496.202} C_VEL
LIN {X 0,Y 323.221,Z 494.165,A -85,B 0,C 180,E1 -15498.05,E2 -15498.05} C_VEL
LIN {X 0,Y 325.472,Z 485.787,A -85,B 0,C 180,E1 -15499.882,E2 -15499.882} C_VEL
LIN {X 0,Y 327.848,Z 476.084,A -85,B 0,C 180,E1 -15501.577,E2 -15501.577} C_VEL
LIN {X 0,Y 329.016,Z 471.026,A -85,B 0,C 180,E1 -15502.328,E2 -15502.328} C_VEL
LIN {X 0,Y 329.152,Z 469.35,A -85,B 0,C 180,E1 -15502.602,E2 -15502.602} C_VEL
LIN {X 0,Y 327.388,Z 462.379,A -85,B 0,C 180,E1 -15504.071,E2 -15504.071} C_VEL
LIN {X 0,Y 323.999,Z 453.138,A -85,B 0,C 180,E1 -15506.111,E2 -15506.111} C_VEL
LIN {X 0,Y 319.762,Z 444.731,A -85,B 0,C 180,E1 -15508.158,E2 -15508.158} C_VEL
LIN {X 0,Y 318.603,Z 442.499,A -85,B 0,C 180,E1 -15508.73,E2 -15508.73} C_VEL
LIN {X 0,Y 316.07,Z 438.523,A -85,B 0,C 180,E1 -15509.866,E2 -15509.866} C_VEL
LIN {X 0,Y 312.925,Z 434.201,A -85,B 0,C 180,E1 -15511.276,E2 -15511.276} C_VEL
LIN {X 0,Y 312.496,Z 432.557,A -85,B 0,C 180,E1 -15511.635,E2 -15511.635} C_VEL
LIN {X 0,Y 312.509,Z 432.557,A -85,B 0,C 180,E1 -15514.21,E2 -15514.21} C_VEL
LIN {X 0,Y 312.528,Z 432.552,A -85,B 0,C 180,E1 -15517.385,E2 -15517.385} C_VEL
LIN {X 0,Y 312.537,Z 432.693,A -85,B 0,C 180,E1 -15520.273,E2 -15520.273} C_VEL
LIN {X 0,Y 314.013,Z 439.769,A -85,B 0,C 180,E1 -15523.933,E2 -15523.933} C_VEL
LIN {X 0,Y 315.485,Z 446.827,A -85,B 0,C 180,E1 -15527.319,E2 -15527.319} C_VEL
LIN {X 0,Y 316.964,Z 454.768,A -85,B 0,C 180,E1 -15530.9,E2 -15530.9} C_VEL
LIN {X 0,Y 317.15,Z 456.516,A -85,B 0,C 180,E1 -15531.649,E2 -15531.649} C_VEL
LIN {X 0,Y 316.33,Z 462.224,A -85,B 0,C 180,E1 -15533.931,E2 -15533.931} C_VEL
LIN {X 0,Y 314.92,Z 471.651,A -85,B 0,C 180,E1 -15537.615,E2 -15537.615} C_VEL
LIN {X 0,Y 314.022,Z 479.267,A -85,B 0,C 180,E1 -15540.48,E2 -15540.48} C_VEL
LIN {X 0,Y 314.732,Z 483.511,A -85,B 0,C 180,E1 -15540.983,E2 -15540.983} C_VEL
LIN {X 0,Y 315.648,Z 486.81,A -85,B 0,C 180,E1 -15541.456,E2 -15541.456} C_VEL
LIN {X 0,Y 316.401,Z 490.927,A -85,B 0,C 180,E1 -15541.959,E2 -15541.959} C_VEL
LIN {X 0,Y 318,Z 499.701,A -85,B 0,C 180,E1 -15543.068,E2 -15543.068} C_VEL
LIN {X 0,Y 319.564,Z 512.496,A -85,B 0,C 180,E1 -15544.627,E2 -15544.627} C_VEL
LIN {X 0,Y 320.279,Z 525.639,A -85,B 0,C 180,E1 -15546.251,E2 -15546.251} C_VEL
LIN {X 0,Y 319.528,Z 537.965,A -85,B 0,C 180,E1 -15547.817,E2 -15547.817} C_VEL
LIN {X 0,Y 318.054,Z 551.542,A -85,B 0,C 180,E1 -15549.802,E2 -15549.802} C_VEL
LIN {X 0,Y 317.199,Z 558.212,A -85,B 0,C 180,E1 -15550.925,E2 -15550.925} C_VEL
LIN {X 0,Y 315.046,Z 568.222,A -85,B 0,C 180,E1 -15552.807,E2 -15552.807} C_VEL
LIN {X 0,Y 313.367,Z 577.079,A -85,B 0,C 180,E1 -15554.844,E2 -15554.844} C_VEL
LIN {X 0,Y 311.933,Z 588.334,A -85,B 0,C 180,E1 -15557.971,E2 -15557.971} C_VEL
LIN {X 0,Y 311.45,Z 594.789,A -85,B 0,C 180,E1 -15560.256,E2 -15560.256} C_VEL
LIN {X 0,Y 311.436,Z 599.045,A -85,B 0,C 180,E1 -15562.218,E2 -15562.218} C_VEL
LIN {X 0,Y 311.57,Z 601.281,A -85,B 0,C 180,E1 -15563.524,E2 -15563.524} C_VEL
LIN {X 0,Y 311.744,Z 603.071,A -85,B 0,C 180,E1 -15564.826,E2 -15564.826} C_VEL
LIN {X 0,Y 311.947,Z 604.445,A -85,B 0,C 180,E1 -15566.124,E2 -15566.124} C_VEL
LIN {X 0,Y 312.033,Z 605.385,A -85,B 0,C 180,E1 -15567.418,E2 -15567.418} C_VEL
LIN {X 0,Y 312.433,Z 605.914,A -85,B 0,C 180,E1 -15568.711,E2 -15568.711} C_VEL
LIN {X 0,Y 312.612,Z 606.002,A -85,B 0,C 180,E1 -15570,E2 -15570} C_VEL
LIN {X 0,Y 312.452,Z 605.636,A -85,B 0,C 180,E1 -15571.289,E2 -15571.289} C_VEL
LIN {X 0,Y 312.087,Z 604.831,A -85,B 0,C 180,E1 -15572.581,E2 -15572.581} C_VEL
LIN {X 0,Y 312,Z 603.602,A -85,B 0,C 180,E1 -15573.875,E2 -15573.875} C_VEL
LIN {X 0,Y 311.717,Z 600.933,A -85,B 0,C 180,E1 -15575.823,E2 -15575.823} C_VEL
LIN {X 0,Y 311.52,Z 597.209,A -85,B 0,C 180,E1 -15577.779,E2 -15577.779} C_VEL
LIN {X 0,Y 311.57,Z 592.358,A -85,B 0,C 180,E1 -15579.74,E2 -15579.74} C_VEL
LIN {X 0,Y 311.98,Z 585.084,A -85,B 0,C 180,E1 -15582.027,E2 -15582.027} C_VEL
LIN {X 0,Y 312.727,Z 577.261,A -85,B 0,C 180,E1 -15583.98,E2 -15583.98} C_VEL
LIN {X 0,Y 313.257,Z 571.552,A -85,B 0,C 180,E1 -15585.166,E2 -15585.166} C_VEL
LIN {X 0,Y 314.496,Z 562.714,A -85,B 0,C 180,E1 -15586.721,E2 -15586.721} C_VEL
LIN {X 0,Y 315.682,Z 552.735,A -85,B 0,C 180,E1 -15588.16,E2 -15588.16} C_VEL
LIN {X 0,Y 315.752,Z 541.565,A -85,B 0,C 180,E1 -15589.504,E2 -15589.504} C_VEL
LIN {X 0,Y 315.556,Z 529.002,A -85,B 0,C 180,E1 -15590.704,E2 -15590.704} C_VEL
LIN {X 0,Y 314.921,Z 517.112,A -85,B 0,C 180,E1 -15591.606,E2 -15591.606} C_VEL
LIN {X 0,Y 313.582,Z 504.096,A -85,B 0,C 180,E1 -15592.374,E2 -15592.374} C_VEL
LIN {X 0,Y 312.179,Z 493.916,A -85,B 0,C 180,E1 -15592.839,E2 -15592.839} C_VEL
LIN {X 0,Y 313.147,Z 481.794,A -85,B 0,C 180,E1 -15597.392,E2 -15597.392} C_VEL
LIN {X 0,Y 314.5,Z 469.939,A -85,B 0,C 180,E1 -15601.878,E2 -15601.878} C_VEL
LIN {X 0,Y 315.925,Z 458.905,A -85,B 0,C 180,E1 -15606.114,E2 -15606.114} C_VEL
LIN {X 0,Y 316.503,Z 454.011,A -85,B 0,C 180,E1 -15608.038,E2 -15608.038} C_VEL
LIN {X 0,Y 315.528,Z 447.595,A -85,B 0,C 180,E1 -15610.772,E2 -15610.772} C_VEL
LIN {X 0,Y 314.002,Z 439.882,A -85,B 0,C 180,E1 -15614.256,E2 -15614.256} C_VEL
LIN {X 0,Y 312.51,Z 432.564,A -85,B 0,C 180,E1 -15617.8,E2 -15617.8} C_VEL
LIN {X 0,Y 312.536,Z 432.556,A -85,B 0,C 180,E1 -15621.91,E2 -15621.91} C_VEL
LIN {X 0,Y 312.507,Z 432.558,A -85,B 0,C 180,E1 -15625.79,E2 -15625.79} C_VEL
LIN {X 0,Y 312.521,Z 432.555,A -85,B 0,C 180,E1 -15628.854,E2 -15628.854} C_VEL
LIN {X 0,Y 312.57,Z 432.55,A -85,B 0,C 180,E1 -15631.824,E2 -15631.824} C_VEL
LIN {X 0,Y 312.586,Z 432.547,A -85,B 0,C 180,E1 -15634.711,E2 -15634.711} C_VEL
LIN {X 0,Y 312.588,Z 432.546,A -85,B 0,C 180,E1 -15637.529,E2 -15637.529} C_VEL
LIN {X 0,Y 312.639,Z 432.541,A -85,B 0,C 180,E1 -15641.657,E2 -15641.657} C_VEL
LIN {X 0,Y 312.695,Z 432.534,A -85,B 0,C 180,E1 -15645.686,E2 -15645.686} C_VEL
LIN {X 0,Y 312.7,Z 432.533,A -85,B 0,C 180,E1 -15649.642,E2 -15649.642} C_VEL
LIN {X 0,Y 312.895,Z 432.508,A -85,B 0,C 180,E1 -15653.552,E2 -15653.552} C_VEL
LIN {X 0,Y 312.94,Z 432.502,A -85,B 0,C 180,E1 -15657.426,E2 -15657.426} C_VEL
LIN {X 0,Y 313.121,Z 432.484,A -85,B 0,C 180,E1 -15660,E2 -15660} C_VEL
LIN {X 0,Y 312.937,Z 432.502,A -85,B 0,C 180,E1 -15662.575,E2 -15662.575} C_VEL
LIN {X 0,Y 312.895,Z 432.505,A -85,B 0,C 180,E1 -15666.652,E2 -15666.652} C_VEL
LIN {X 0,Y 312.788,Z 432.52,A -85,B 0,C 180,E1 -15669.049,E2 -15669.049} C_VEL
LIN {X 0,Y 312.635,Z 432.536,A -85,B 0,C 180,E1 -15672.991,E2 -15672.991} C_VEL
LIN {X 0,Y 312.639,Z 432.54,A -85,B 0,C 180,E1 -15675.65,E2 -15675.65} C_VEL
LIN {X 0,Y 312.632,Z 432.537,A -85,B 0,C 180,E1 -15679.237,E2 -15679.237} C_VEL
LIN {X 0,Y 312.547,Z 432.542,A -85,B 0,C 180,E1 -15682.79,E2 -15682.79} C_VEL
LIN {X 0,Y 312.603,Z 432.546,A -85,B 0,C 180,E1 -15685.936,E2 -15685.936} C_VEL
LIN {X 0,Y 312.539,Z 432.554,A -85,B 0,C 180,E1 -15689.651,E2 -15689.651} C_VEL
LIN {X 0,Y 312.521,Z 432.549,A -85,B 0,C 180,E1 -15693.689,E2 -15693.689} C_VEL
LIN {X 0,Y 312.539,Z 432.552,A -85,B 0,C 180,E1 -15697.384,E2 -15697.384} C_VEL
LIN {X 0,Y 312.491,Z 432.556,A -85,B 0,C 180,E1 -15700.709,E2 -15700.709} C_VEL
LIN {X 0,Y 312.454,Z 432.562,A -85,B 0,C 180,E1 -15704.21,E2 -15704.21} C_VEL
LIN {X 0,Y 312.486,Z 432.56,A -85,B 0,C 180,E1 -15707.919,E2 -15707.919} C_VEL
LIN {X 0,Y 312.537,Z 432.554,A -85,B 0,C 180,E1 -15711.911,E2 -15711.911} C_VEL
LIN {X 0,Y 312.509,Z 432.559,A -85,B 0,C 180,E1 -15715.79,E2 -15715.79} C_VEL
LIN {X 0,Y 312.531,Z 432.552,A -85,B 0,C 180,E1 -15718.855,E2 -15718.855} C_VEL
LIN {X 0,Y 312.588,Z 432.547,A -85,B 0,C 180,E1 -15721.826,E2 -15721.826} C_VEL
LIN {X 0,Y 312.588,Z 432.544,A -85,B 0,C 180,E1 -15724.711,E2 -15724.711} C_VEL
LIN {X 0,Y 312.59,Z 432.549,A -85,B 0,C 180,E1 -15727.529,E2 -15727.529} C_VEL
LIN {X 0,Y 312.67,Z 432.538,A -85,B 0,C 180,E1 -15731.296,E2 -15731.296} C_VEL
LIN {X 0,Y 316.762,Z 444.684,A -85,B 0,C 180,E1 -15732.563,E2 -15732.563} C_VEL
LIN {X 0,Y 319.87,Z 455.514,A -85,B 0,C 180,E1 -15733.896,E2 -15733.896} C_VEL
LIN {X 0,Y 320.451,Z 458.14,A -85,B 0,C 180,E1 -15734.252,E2 -15734.252} C_VEL
LIN {X 0,Y 319.32,Z 468.972,A -85,B 0,C 180,E1 -15735.632,E2 -15735.632} C_VEL
LIN {X 0,Y 318.045,Z 478.956,A -85,B 0,C 180,E1 -15737.234,E2 -15737.234} C_VEL
LIN {X 0,Y 316.887,Z 486.963,A -85,B 0,C 180,E1 -15738.81,E2 -15738.81} C_VEL
LIN {X 0,Y 315.729,Z 494.8,A -85,B 0,C 180,E1 -15740.713,E2 -15740.713} C_VEL
LIN {X 0,Y 314.901,Z 500.112,A -85,B 0,C 180,E1 -15742.305,E2 -15742.305} C_VEL
LIN {X 0,Y 314.28,Z 505.278,A -85,B 0,C 180,E1 -15744.225,E2 -15744.225} C_VEL
LIN {X 0,Y 313.541,Z 509.35,A -85,B 0,C 180,E1 -15746.145,E2 -15746.145} C_VEL
LIN {X 0,Y 313.183,Z 511.507,A -85,B 0,C 180,E1 -15747.428,E2 -15747.428} C_VEL
LIN {X 0,Y 312.849,Z 514.458,A -85,B 0,C 180,E1 -15750,E2 -15750} C_VEL
LIN {X 0,Y 312.83,Z 515.351,A -85,B 0,C 180,E1 -15751.288,E2 -15751.288} C_VEL
LIN {X 0,Y 312.716,Z 515.886,A -85,B 0,C 180,E1 -15752.576,E2 -15752.576} C_VEL
LIN {X 0,Y 312.611,Z 516.011,A -85,B 0,C 180,E1 -15753.868,E2 -15753.868} C_VEL
LIN {X 0,Y 313.078,Z 515.076,A -85,B 0,C 180,E1 -15756.445,E2 -15756.445} C_VEL
LIN {X 0,Y 313.506,Z 514.026,A -85,B 0,C 180,E1 -15757.73,E2 -15757.73} C_VEL
LIN {X 0,Y 314.185,Z 510.886,A -85,B 0,C 180,E1 -15760.185,E2 -15760.185} C_VEL
LIN {X 0,Y 315.069,Z 507.034,A -85,B 0,C 180,E1 -15762.235,E2 -15762.235} C_VEL
LIN {X 0,Y 315.913,Z 502.293,A -85,B 0,C 180,E1 -15764.165,E2 -15764.165} C_VEL
LIN {X 0,Y 317.01,Z 496.286,A -85,B 0,C 180,E1 -15766.089,E2 -15766.089} C_VEL
LIN {X 0,Y 318.346,Z 488.761,A -85,B 0,C 180,E1 -15768.004,E2 -15768.004} C_VEL
LIN {X 0,Y 319.685,Z 481.013,A -85,B 0,C 180,E1 -15769.589,E2 -15769.589} C_VEL
LIN {X 0,Y 320.973,Z 471.546,A -85,B 0,C 180,E1 -15771.179,E2 -15771.179} C_VEL
LIN {X 0,Y 322.228,Z 461.155,A -85,B 0,C 180,E1 -15772.585,E2 -15772.585} C_VEL
LIN {X 0,Y 319.079,Z 450.36,A -85,B 0,C 180,E1 -15774.121,E2 -15774.121} C_VEL
LIN {X 0,Y 315.268,Z 439.601,A -85,B 0,C 180,E1 -15775.448,E2 -15775.448} C_VEL
LIN {X 0,Y 312.644,Z 432.91,A -85,B 0,C 180,E1 -15776.184,E2 -15776.184} C_VEL
LIN {X 0,Y 312.58,Z 432.549,A -85,B 0,C 180,E1 -15776.261,E2 -15776.261} C_VEL
LIN {X 0,Y 312.549,Z 432.551,A -85,B 0,C 180,E1 -15779.65,E2 -15779.65} C_VEL
LIN {X 0,Y 312.523,Z 432.555,A -85,B 0,C 180,E1 -15783.689,E2 -15783.689} C_VEL
LIN {X 0,Y 312.541,Z 432.552,A -85,B 0,C 180,E1 -15787.383,E2 -15787.383} C_VEL
LIN {X 0,Y 312.494,Z 432.558,A -85,B 0,C 180,E1 -15790.709,E2 -15790.709} C_VEL
LIN {X 0,Y 312.455,Z 432.565,A -85,B 0,C 180,E1 -15794.21,E2 -15794.21} C_VEL
LIN {X 0,Y 312.488,Z 432.56,A -85,B 0,C 180,E1 -15797.919,E2 -15797.919} C_VEL
LIN {X 0,Y 312.538,Z 432.555,A -85,B 0,C 180,E1 -15801.91,E2 -15801.91} C_VEL
LIN {X 0,Y 312.51,Z 432.558,A -85,B 0,C 180,E1 -15805.79,E2 -15805.79} C_VEL
LIN {X 0,Y 312.528,Z 432.552,A -85,B 0,C 180,E1 -15808.854,E2 -15808.854} C_VEL
LIN {X 0,Y 312.578,Z 432.549,A -85,B 0,C 180,E1 -15811.825,E2 -15811.825} C_VEL
LIN {X 0,Y 312.589,Z 432.544,A -85,B 0,C 180,E1 -15814.711,E2 -15814.711} C_VEL
LIN {X 0,Y 312.542,Z 432.55,A -85,B 0,C 180,E1 -15818.913,E2 -15818.913} C_VEL
LIN {X 0,Y 312.705,Z 432.724,A -85,B 0,C 180,E1 -15822.168,E2 -15822.168} C_VEL
LIN {X 0,Y 315.526,Z 444.401,A -85,B 0,C 180,E1 -15823.293,E2 -15823.293} C_VEL
LIN {X 0,Y 316.865,Z 449.745,A -85,B 0,C 180,E1 -15823.889,E2 -15823.889} C_VEL
LIN {X 0,Y 316.584,Z 454.78,A -85,B 0,C 180,E1 -15824.445,E2 -15824.445} C_VEL
LIN {X 0,Y 315.561,Z 459.736,A -85,B 0,C 180,E1 -15825.017,E2 -15825.017} C_VEL
LIN {X 0,Y 312.179,Z 467.502,A -85,B 0,C 180,E1 -15825.967,E2 -15825.967} C_VEL
LIN {X 0,Y 308.802,Z 474.865,A -85,B 0,C 180,E1 -15827.02,E2 -15827.02} C_VEL
LIN {X 0,Y 307.787,Z 479.14,A -85,B 0,C 180,E1 -15827.752,E2 -15827.752} C_VEL
LIN {X 0,Y 307.141,Z 487.635,A -85,B 0,C 180,E1 -15829.452,E2 -15829.452} C_VEL
LIN {X 0,Y 306.49,Z 495.818,A -85,B 0,C 180,E1 -15831.428,E2 -15831.428} C_VEL
LIN {X 0,Y 306.01,Z 502.455,A -85,B 0,C 180,E1 -15833.406,E2 -15833.406} C_VEL
LIN {X 0,Y 305.649,Z 507.847,A -85,B 0,C 180,E1 -15835.384,E2 -15835.384} C_VEL
LIN {X 0,Y 305.503,Z 510.833,A -85,B 0,C 180,E1 -15836.703,E2 -15836.703} C_VEL
LIN {X 0,Y 305.587,Z 514.388,A -85,B 0,C 180,E1 -15838.682,E2 -15838.682} C_VEL
LIN {X 0,Y 305.775,Z 516.18,A -85,B 0,C 180,E1 -15840,E2 -15840} C_VEL
LIN {X 0,Y 306.072,Z 518.605,A -85,B 0,C 180,E1 -15842.632,E2 -15842.632} C_VEL
LIN {X 0,Y 306.365,Z 519.205,A -85,B 0,C 180,E1 -15843.946,E2 -15843.946} C_VEL
LIN {X 0,Y 307.245,Z 519.172,A -85,B 0,C 180,E1 -15846.567,E2 -15846.567} C_VEL
LIN {X 0,Y 307.852,Z 518.57,A -85,B 0,C 180,E1 -15847.873,E2 -15847.873} C_VEL
LIN {X 0,Y 309.396,Z 516.117,A -85,B 0,C 180,E1 -15850.47,E2 -15850.47} C_VEL
LIN {X 0,Y 310.801,Z 513.187,A -85,B 0,C 180,E1 -15852.405,E2 -15852.405} C_VEL
LIN {X 0,Y 312.445,Z 509.215,A -85,B 0,C 180,E1 -15854.325,E2 -15854.325} C_VEL
LIN {X 0,Y 314.319,Z 504.192,A -85,B 0,C 180,E1 -15856.23,E2 -15856.23} C_VEL
LIN {X 0,Y 316.501,Z 497.872,A -85,B 0,C 180,E1 -15858.112,E2 -15858.112} C_VEL
LIN {X 0,Y 319.262,Z 488.644,A -85,B 0,C 180,E1 -15860.286,E2 -15860.286} C_VEL
LIN {X 0,Y 321.871,Z 479.104,A -85,B 0,C 180,E1 -15862.054,E2 -15862.054} C_VEL
LIN {X 0,Y 323.359,Z 472.884,A -85,B 0,C 180,E1 -15863.03,E2 -15863.03} C_VEL
LIN {X 0,Y 322.004,Z 466.312,A -85,B 0,C 180,E1 -15864.5,E2 -15864.5} C_VEL
LIN {X 0,Y 319.076,Z 457.619,A -85,B 0,C 180,E1 -15866.545,E2 -15866.545} C_VEL
LIN {X 0,Y 315.645,Z 450.214,A -85,B 0,C 180,E1 -15868.478,E2 -15868.478} C_VEL
LIN {X 0,Y 312.03,Z 443.83,A -85,B 0,C 180,E1 -15870.374,E2 -15870.374} C_VEL
LIN {X 0,Y 309.382,Z 439.81,A -85,B 0,C 180,E1 -15871.752,E2 -15871.752} C_VEL
LIN {X 0,Y 308.918,Z 438.695,A -85,B 0,C 180,E1 -15872.063,E2 -15872.063} C_VEL
LIN {X 0,Y 306.858,Z 436.857,A -85,B 0,C 180,E1 -15873.057,E2 -15873.057} C_VEL
LIN {X 0,Y 305.967,Z 435.214,A -85,B 0,C 180,E1 -15873.678,E2 -15873.678} C_VEL
LIN {X 0,Y 305.774,Z 434.799,A -85,B 0,C 180,E1 -15876.698,E2 -15876.698} C_VEL
LIN {X 0,Y 305.9,Z 435.054,A -85,B 0,C 180,E1 -15880.038,E2 -15880.038} C_VEL
LIN {X 0,Y 305.874,Z 435.44,A -85,B 0,C 180,E1 -15880.691,E2 -15880.691} C_VEL
LIN {X 0,Y 307.235,Z 441.99,A -85,B 0,C 180,E1 -15884.135,E2 -15884.135} C_VEL
LIN {X 0,Y 308.736,Z 449.329,A -85,B 0,C 180,E1 -15887.715,E2 -15887.715} C_VEL
LIN {X 0,Y 309.926,Z 455.54,A -85,B 0,C 180,E1 -15890.584,E2 -15890.584} C_VEL
LIN {X 0,Y 310.15,Z 457.512,A -85,B 0,C 180,E1 -15891.453,E2 -15891.453} C_VEL
LIN {X 0,Y 309.351,Z 463.199,A -85,B 0,C 180,E1 -15893.794,E2 -15893.794} C_VEL
LIN {X 0,Y 307.835,Z 472.804,A -85,B 0,C 180,E1 -15897.642,E2 -15897.642} C_VEL
LIN {X 0,Y 307.549,Z 475.355,A -85,B 0,C 180,E1 -15898.604,E2 -15898.604} C_VEL
LIN {X 0,Y 308.289,Z 480.097,A -85,B 0,C 180,E1 -15899.241,E2 -15899.241} C_VEL
LIN {X 0,Y 309.366,Z 483.579,A -85,B 0,C 180,E1 -15899.826,E2 -15899.826} C_VEL
LIN {X 0,Y 311.784,Z 497.47,A -85,B 0,C 180,E1 -15901.747,E2 -15901.747} C_VEL
LIN {X 0,Y 313.202,Z 507.878,A -85,B 0,C 180,E1 -15903.136,E2 -15903.136} C_VEL
LIN {X 0,Y 314.031,Z 522.174,A -85,B 0,C 180,E1 -15905.012,E2 -15905.012} C_VEL
LIN {X 0,Y 313.853,Z 532.349,A -85,B 0,C 180,E1 -15906.38,E2 -15906.38} C_VEL
LIN {X 0,Y 312.234,Z 546.24,A -85,B 0,C 180,E1 -15908.371,E2 -15908.371} C_VEL
LIN {X 0,Y 310.513,Z 558.686,A -85,B 0,C 180,E1 -15910.497,E2 -15910.497} C_VEL
LIN {X 0,Y 308.257,Z 568.312,A -85,B 0,C 180,E1 -15912.417,E2 -15912.417} C_VEL
LIN {X 0,Y 306.364,Z 577.398,A -85,B 0,C 180,E1 -15914.637,E2 -15914.637} C_VEL
LIN {X 0,Y 304.938,Z 587.401,A -85,B 0,C 180,E1 -15917.69,E2 -15917.69} C_VEL
LIN {X 0,Y 304.38,Z 593.824,A -85,B 0,C 180,E1 -15920.027,E2 -15920.027} C_VEL
LIN {X 0,Y 304.365,Z 598.071,A -85,B 0,C 180,E1 -15922.036,E2 -15922.036} C_VEL
LIN {X 0,Y 304.496,Z 600.295,A -85,B 0,C 180,E1 -15923.373,E2 -15923.373} C_VEL
LIN {X 0,Y 304.657,Z 602.078,A -85,B 0,C 180,E1 -15924.705,E2 -15924.705} C_VEL
LIN {X 0,Y 304.897,Z 603.452,A -85,B 0,C 180,E1 -15926.034,E2 -15926.034} C_VEL
LIN {X 0,Y 304.986,Z 604.382,A -85,B 0,C 180,E1 -15927.358,E2 -15927.358} C_VEL
LIN {X 0,Y 305.396,Z 604.904,A -85,B 0,C 180,E1 -15928.681,E2 -15928.681} C_VEL
LIN {X 0,Y 305.603,Z 604.989,A -85,B 0,C 180,E1 -15930,E2 -15930} C_VEL
LIN {X 0,Y 305.417,Z 604.612,A -85,B 0,C 180,E1 -15931.318,E2 -15931.318} C_VEL
LIN {X 0,Y 305.041,Z 603.794,A -85,B 0,C 180,E1 -15932.641,E2 -15932.641} C_VEL
LIN {X 0,Y 304.953,Z 602.553,A -85,B 0,C 180,E1 -15933.964,E2 -15933.964} C_VEL
LIN {X 0,Y 304.635,Z 599.859,A -85,B 0,C 180,E1 -15935.959,E2 -15935.959} C_VEL
LIN {X 0,Y 304.448,Z 596.117,A -85,B 0,C 180,E1 -15937.961,E2 -15937.961} C_VEL
LIN {X 0,Y 304.496,Z 591.241,A -85,B 0,C 180,E1 -15939.968,E2 -15939.968} C_VEL
LIN {X 0,Y 304.977,Z 583.951,A -85,B 0,C 180,E1 -15942.307,E2 -15942.307} C_VEL
LIN {X 0,Y 305.731,Z 576.094,A -85,B 0,C 180,E1 -15944.307,E2 -15944.307} C_VEL
LIN {X 0,Y 306.415,Z 570.383,A -85,B 0,C 180,E1 -15945.513,E2 -15945.513} C_VEL
LIN {X 0,Y 307.617,Z 561.499,A -85,B 0,C 180,E1 -15947.106,E2 -15947.106} C_VEL
LIN {X 0,Y 308.676,Z 552.673,A -85,B 0,C 180,E1 -15948.415,E2 -15948.415} C_VEL
LIN {X 0,Y 308.828,Z 541.757,A -85,B 0,C 180,E1 -15949.786,E2 -15949.786} C_VEL
LIN {X 0,Y 308.685,Z 529.556,A -85,B 0,C 180,E1 -15951.018,E2 -15951.018} C_VEL
LIN {X 0,Y 308.05,Z 517.136,A -85,B 0,C 180,E1 -15952.008,E2 -15952.008} C_VEL
LIN {X 0,Y 306.769,Z 504.171,A -85,B 0,C 180,E1 -15952.812,E2 -15952.812} C_VEL
LIN {X 0,Y 305.171,Z 492.853,A -85,B 0,C 180,E1 -15953.371,E2 -15953.371} C_VEL
LIN {X 0,Y 306.048,Z 482.578,A -85,B 0,C 180,E1 -15957.34,E2 -15957.34} C_VEL
LIN {X 0,Y 307.364,Z 471.265,A -85,B 0,C 180,E1 -15961.729,E2 -15961.729} C_VEL
LIN {X 0,Y 308.598,Z 461.672,A -85,B 0,C 180,E1 -15965.509,E2 -15965.509} C_VEL
LIN {X 0,Y 309.499,Z 455.896,A -85,B 0,C 180,E1 -15967.814,E2 -15967.814} C_VEL
LIN {X 0,Y 309.104,Z 451.849,A -85,B 0,C 180,E1 -15969.541,E2 -15969.541} C_VEL
LIN {X 0,Y 307.552,Z 443.588,A -85,B 0,C 180,E1 -15973.278,E2 -15973.278} C_VEL
LIN {X 0,Y 305.812,Z 435.289,A -85,B 0,C 180,E1 -15977.341,E2 -15977.341} C_VEL
LIN {X 0,Y 305.443,Z 433.442,A -85,B 0,C 180,E1 -15978.316,E2 -15978.316} C_VEL
LIN {X 0,Y 305.496,Z 433.431,A -85,B 0,C 180,E1 -15981.601,E2 -15981.601} C_VEL
LIN {X 0,Y 305.463,Z 433.435,A -85,B 0,C 180,E1 -15984.887,E2 -15984.887} C_VEL
LIN {X 0,Y 305.45,Z 433.44,A -85,B 0,C 180,E1 -15988.355,E2 -15988.355} C_VEL
LIN {X 0,Y 305.513,Z 433.427,A -85,B 0,C 180,E1 -15991.113,E2 -15991.113} C_VEL
LIN {X 0,Y 305.571,Z 433.423,A -85,B 0,C 180,E1 -15994.088,E2 -15994.088} C_VEL
LIN {X 0,Y 305.528,Z 433.429,A -85,B 0,C 180,E1 -15998.405,E2 -15998.405} C_VEL
LIN {X 0,Y 305.591,Z 433.418,A -85,B 0,C 180,E1 -16001.218,E2 -16001.218} C_VEL
LIN {X 0,Y 305.65,Z 433.41,A -85,B 0,C 180,E1 -16005.349,E2 -16005.349} C_VEL
LIN {X 0,Y 305.638,Z 433.412,A -85,B 0,C 180,E1 -16009.4,E2 -16009.4} C_VEL
LIN {X 0,Y 305.774,Z 433.399,A -85,B 0,C 180,E1 -16012.073,E2 -16012.073} C_VEL
LIN {X 0,Y 305.688,Z 433.405,A -85,B 0,C 180,E1 -16014.724,E2 -16014.724} C_VEL
LIN {X 0,Y 305.959,Z 433.371,A -85,B 0,C 180,E1 -16018.684,E2 -16018.684} C_VEL
LIN {X 0,Y 305.958,Z 433.37,A -85,B 0,C 180,E1 -16021.316,E2 -16021.316} C_VEL
LIN {X 0,Y 305.854,Z 433.382,A -85,B 0,C 180,E1 -16026.598,E2 -16026.598} C_VEL
LIN {X 0,Y 305.737,Z 433.398,A -85,B 0,C 180,E1 -16029.26,E2 -16029.26} C_VEL
LIN {X 0,Y 305.59,Z 433.413,A -85,B 0,C 180,E1 -16033.296,E2 -16033.296} C_VEL
LIN {X 0,Y 305.595,Z 433.42,A -85,B 0,C 180,E1 -16036.02,E2 -16036.02} C_VEL
LIN {X 0,Y 305.578,Z 433.416,A -85,B 0,C 180,E1 -16039.445,E2 -16039.445} C_VEL
LIN {X 0,Y 305.491,Z 433.419,A -85,B 0,C 180,E1 -16043.042,E2 -16043.042} C_VEL
LIN {X 0,Y 305.548,Z 433.424,A -85,B 0,C 180,E1 -16046.227,E2 -16046.227} C_VEL
LIN {X 0,Y 305.489,Z 433.429,A -85,B 0,C 180,E1 -16049.048,E2 -16049.048} C_VEL
LIN {X 0,Y 305.444,Z 433.431,A -85,B 0,C 180,E1 -16051.953,E2 -16051.953} C_VEL
LIN {X 0,Y 305.464,Z 433.429,A -85,B 0,C 180,E1 -16055.113,E2 -16055.113} C_VEL
LIN {X 0,Y 305.468,Z 433.432,A -85,B 0,C 180,E1 -16058.533,E2 -16058.533} C_VEL
LIN {X 0,Y 305.457,Z 433.433,A -85,B 0,C 180,E1 -16062.586,E2 -16062.586} C_VEL
LIN {X 0,Y 305.428,Z 433.437,A -85,B 0,C 180,E1 -16066.345,E2 -16066.345} C_VEL
LIN {X 0,Y 305.46,Z 433.436,A -85,B 0,C 180,E1 -16069.893,E2 -16069.893} C_VEL
LIN {X 0,Y 305.501,Z 433.43,A -85,B 0,C 180,E1 -16073.627,E2 -16073.627} C_VEL
LIN {X 0,Y 305.468,Z 433.431,A -85,B 0,C 180,E1 -16076.484,E2 -16076.484} C_VEL
LIN {X 0,Y 305.471,Z 433.435,A -85,B 0,C 180,E1 -16079.592,E2 -16079.592} C_VEL
LIN {X 0,Y 305.543,Z 433.423,A -85,B 0,C 180,E1 -16082.611,E2 -16082.611} C_VEL
LIN {X 0,Y 305.511,Z 433.428,A -85,B 0,C 180,E1 -16085.539,E2 -16085.539} C_VEL
LIN {X 0,Y 305.524,Z 433.429,A -85,B 0,C 180,E1 -16089.816,E2 -16089.816} C_VEL
LIN {X 0,Y 305.633,Z 433.593,A -85,B 0,C 180,E1 -16090.815,E2 -16090.815} C_VEL
LIN {X 0,Y 309.403,Z 444.489,A -85,B 0,C 180,E1 -16091.972,E2 -16091.972} C_VEL
LIN {X 0,Y 312.713,Z 455.505,A -85,B 0,C 180,E1 -16093.349,E2 -16093.349} C_VEL
LIN {X 0,Y 313.689,Z 459.497,A -85,B 0,C 180,E1 -16093.904,E2 -16093.904} C_VEL
LIN {X 0,Y 312.494,Z 470.46,A -85,B 0,C 180,E1 -16095.345,E2 -16095.345} C_VEL
LIN {X 0,Y 311.22,Z 480.177,A -85,B 0,C 180,E1 -16096.949,E2 -16096.949} C_VEL
LIN {X 0,Y 310.018,Z 488.15,A -85,B 0,C 180,E1 -16098.559,E2 -16098.559} C_VEL
LIN {X 0,Y 308.821,Z 495.956,A -85,B 0,C 180,E1 -16100.503,E2 -16100.503} C_VEL
LIN {X 0,Y 307.967,Z 501.241,A -85,B 0,C 180,E1 -16102.13,E2 -16102.13} C_VEL
LIN {X 0,Y 307.306,Z 506.384,A -85,B 0,C 180,E1 -16104.093,E2 -16104.093} C_VEL
LIN {X 0,Y 306.539,Z 510.436,A -85,B 0,C 180,E1 -16106.056,E2 -16106.056} C_VEL
LIN {X 0,Y 306.167,Z 512.576,A -85,B 0,C 180,E1 -16107.369,E2 -16107.369} C_VEL
LIN {X 0,Y 305.824,Z 515.503,A -85,B 0,C 180,E1 -16110,E2 -16110} C_VEL
LIN {X 0,Y 305.808,Z 516.387,A -85,B 0,C 180,E1 -16111.317,E2 -16111.317} C_VEL
LIN {X 0,Y 305.693,Z 516.905,A -85,B 0,C 180,E1 -16112.636,E2 -16112.636} C_VEL
LIN {X 0,Y 305.591,Z 517.019,A -85,B 0,C 180,E1 -16113.957,E2 -16113.957} C_VEL
LIN {X 0,Y 306.091,Z 516.065,A -85,B 0,C 180,E1 -16116.593,E2 -16116.593} C_VEL
LIN {X 0,Y 306.538,Z 514.998,A -85,B 0,C 180,E1 -16117.907,E2 -16117.907} C_VEL
LIN {X 0,Y 307.27,Z 511.835,A -85,B 0,C 180,E1 -16120.416,E2 -16120.416} C_VEL
LIN {X 0,Y 308.199,Z 507.96,A -85,B 0,C 180,E1 -16122.512,E2 -16122.512} C_VEL
LIN {X 0,Y 309.078,Z 503.199,A -85,B 0,C 180,E1 -16124.485,E2 -16124.485} C_VEL
LIN {X 0,Y 310.226,Z 497.168,A -85,B 0,C 180,E1 -16126.45,E2 -16126.45} C_VEL
LIN {X 0,Y 311.657,Z 489.595,A -85,B 0,C 180,E1 -16128.404,E2 -16128.404} C_VEL
LIN {X 0,Y 313.046,Z 481.813,A -85,B 0,C 180,E1 -16130.022,E2 -16130.022} C_VEL
LIN {X 0,Y 314.39,Z 472.304,A -85,B 0,C 180,E1 -16131.645,E2 -16131.645} C_VEL
LIN {X 0,Y 315.49,Z 462.763,A -85,B 0,C 180,E1 -16132.974,E2 -16132.974} C_VEL
LIN {X 0,Y 312.588,Z 452.692,A -85,B 0,C 180,E1 -16134.472,E2 -16134.472} C_VEL
LIN {X 0,Y 308.846,Z 442.029,A -85,B 0,C 180,E1 -16135.858,E2 -16135.858} C_VEL
LIN {X 0,Y 305.523,Z 433.426,A -85,B 0,C 180,E1 -16136.857,E2 -16136.857} C_VEL
LIN {X 0,Y 305.468,Z 433.436,A -85,B 0,C 180,E1 -16140.409,E2 -16140.409} C_VEL
LIN {X 0,Y 305.468,Z 433.436,A -85,B 0,C 180,E1 -16144.079,E2 -16144.079} C_VEL
LIN {X 0,Y 305.499,Z 433.43,A -85,B 0,C 180,E1 -16146.737,E2 -16146.737} C_VEL
LIN {X 0,Y 305.458,Z 433.435,A -85,B 0,C 180,E1 -16150.6,E2 -16150.6} C_VEL
LIN {X 0,Y 305.429,Z 433.439,A -85,B 0,C 180,E1 -16153.655,E2 -16153.655} C_VEL
LIN {X 0,Y 305.459,Z 433.432,A -85,B 0,C 180,E1 -16157.414,E2 -16157.414} C_VEL
LIN {X 0,Y 305.498,Z 433.429,A -85,B 0,C 180,E1 -16161.6,E2 -16161.6} C_VEL
LIN {X 0,Y 305.466,Z 433.431,A -85,B 0,C 180,E1 -16164.887,E2 -16164.887} C_VEL
LIN {X 0,Y 305.456,Z 433.435,A -85,B 0,C 180,E1 -16168.355,E2 -16168.355} C_VEL
LIN {X 0,Y 305.524,Z 433.425,A -85,B 0,C 180,E1 -16171.114,E2 -16171.114} C_VEL
LIN {X 0,Y 305.575,Z 433.421,A -85,B 0,C 180,E1 -16174.088,E2 -16174.088} C_VEL
LIN {X 0,Y 305.486,Z 433.43,A -85,B 0,C 180,E1 -16178.401,E2 -16178.401} C_VEL
LIN {X 0,Y 305.656,Z 433.559,A -85,B 0,C 180,E1 -16181.959,E2 -16181.959} C_VEL
LIN {X 0,Y 308.484,Z 445.33,A -85,B 0,C 180,E1 -16183.111,E2 -16183.111} C_VEL
LIN {X 0,Y 309.904,Z 451.212,A -85,B 0,C 180,E1 -16183.783,E2 -16183.783} C_VEL
LIN {X 0,Y 308.983,Z 463.97,A -85,B 0,C 180,E1 -16185.342,E2 -16185.342} C_VEL
LIN {X 0,Y 308.285,Z 473.791,A -85,B 0,C 180,E1 -16186.822,E2 -16186.822} C_VEL
LIN {X 0,Y 307.787,Z 479.14,A -85,B 0,C 180,E1 -16187.752,E2 -16187.752} C_VEL
LIN {X 0,Y 306.763,Z 483.295,A -85,B 0,C 180,E1 -16188.519,E2 -16188.519} C_VEL
LIN {X 0,Y 303.365,Z 489.716,A -85,B 0,C 180,E1 -16189.792,E2 -16189.792} C_VEL
LIN {X 0,Y 300.077,Z 495.682,A -85,B 0,C 180,E1 -16191.169,E2 -16191.169} C_VEL
LIN {X 0,Y 299.242,Z 499.043,A -85,B 0,C 180,E1 -16192.081,E2 -16192.081} C_VEL
LIN {X 0,Y 298.887,Z 504.821,A -85,B 0,C 180,E1 -16193.926,E2 -16193.926} C_VEL
LIN {X 0,Y 298.378,Z 509.987,A -85,B 0,C 180,E1 -16195.948,E2 -16195.948} C_VEL
LIN {X 0,Y 298.549,Z 514.014,A -85,B 0,C 180,E1 -16197.976,E2 -16197.976} C_VEL
LIN {X 0,Y 298.75,Z 517.046,A -85,B 0,C 180,E1 -16200,E2 -16200} C_VEL
LIN {X 0,Y 299.06,Z 519.632,A -85,B 0,C 180,E1 -16202.694,E2 -16202.694} C_VEL
LIN {X 0,Y 299.372,Z 520.344,A -85,B 0,C 180,E1 -16204.038,E2 -16204.038} C_VEL
LIN {X 0,Y 299.784,Z 520.627,A -85,B 0,C 180,E1 -16205.381,E2 -16205.381} C_VEL
LIN {X 0,Y 300.965,Z 520.002,A -85,B 0,C 180,E1 -16208.054,E2 -16208.054} C_VEL
LIN {X 0,Y 301.782,Z 519.096,A -85,B 0,C 180,E1 -16209.382,E2 -16209.382} C_VEL
LIN {X 0,Y 303.558,Z 516.022,A -85,B 0,C 180,E1 -16212.027,E2 -16212.027} C_VEL
LIN {X 0,Y 305.297,Z 512.607,A -85,B 0,C 180,E1 -16213.987,E2 -16213.987} C_VEL
LIN {X 0,Y 307.177,Z 508.164,A -85,B 0,C 180,E1 -16215.935,E2 -16215.935} C_VEL
LIN {X 0,Y 309.715,Z 501.444,A -85,B 0,C 180,E1 -16218.18,E2 -16218.18} C_VEL
LIN {X 0,Y 312.228,Z 494.297,A -85,B 0,C 180,E1 -16220.076,E2 -16220.076} C_VEL
LIN {X 0,Y 314.932,Z 485.45,A -85,B 0,C 180,E1 -16221.95,E2 -16221.95} C_VEL
LIN {X 0,Y 317.609,Z 475.371,A -85,B 0,C 180,E1 -16223.697,E2 -16223.697} C_VEL
LIN {X 0,Y 315.86,Z 467.585,A -85,B 0,C 180,E1 -16225.592,E2 -16225.592} C_VEL
LIN {X 0,Y 313.678,Z 460.923,A -85,B 0,C 180,E1 -16227.312,E2 -16227.312} C_VEL
LIN {X 0,Y 310.784,Z 454.267,A -85,B 0,C 180,E1 -16229.203,E2 -16229.203} C_VEL
LIN {X 0,Y 307.626,Z 448.625,A -85,B 0,C 180,E1 -16231.067,E2 -16231.067} C_VEL
LIN {X 0,Y 305.855,Z 445.486,A -85,B 0,C 180,E1 -16232.192,E2 -16232.192} C_VEL
LIN {X 0,Y 303.216,Z 442.005,A -85,B 0,C 180,E1 -16233.799,E2 -16233.799} C_VEL
LIN {X 0,Y 299.809,Z 438.651,A -85,B 0,C 180,E1 -16236.059,E2 -16236.059} C_VEL
LIN {X 0,Y 299.911,Z 438.877,A -85,B 0,C 180,E1 -16239.347,E2 -16239.347} C_VEL
LIN {X 0,Y 299.691,Z 440.316,A -85,B 0,C 180,E1 -16242.307,E2 -16242.307} C_VEL
LIN {X 0,Y 301.241,Z 448.1,A -85,B 0,C 180,E1 -16246.322,E2 -16246.322} C_VEL
LIN {X 0,Y 302.748,Z 455.785,A -85,B 0,C 180,E1 -16250.002,E2 -16250.002} C_VEL
LIN {X 0,Y 303.141,Z 458.512,A -85,B 0,C 180,E1 -16251.246,E2 -16251.246} C_VEL
LIN {X 0,Y 302.716,Z 462.288,A -85,B 0,C 180,E1 -16252.869,E2 -16252.869} C_VEL
LIN {X 0,Y 301.321,Z 470.744,A -85,B 0,C 180,E1 -16256.319,E2 -16256.319} C_VEL
LIN {X 0,Y 301.829,Z 474.946,A -85,B 0,C 180,E1 -16256.956,E2 -16256.956} C_VEL
LIN {X 0,Y 303.017,Z 479.047,A -85,B 0,C 180,E1 -16257.761,E2 -16257.761} C_VEL
LIN {X 0,Y 304.116,Z 485.388,A -85,B 0,C 180,E1 -16258.766,E2 -16258.766} C_VEL
LIN {X 0,Y 304.632,Z 487.014,A -85,B 0,C 180,E1 -16259.076,E2 -16259.076} C_VEL
LIN {X 0,Y 307.065,Z 504.851,A -85,B 0,C 180,E1 -16261.703,E2 -16261.703} C_VEL
LIN {X 0,Y 307.913,Z 518.68,A -85,B 0,C 180,E1 -16263.652,E2 -16263.652} C_VEL
LIN {X 0,Y 307.836,Z 530.704,A -85,B 0,C 180,E1 -16265.376,E2 -16265.376} C_VEL
LIN {X 0,Y 306.206,Z 544.242,A -85,B 0,C 180,E1 -16267.39,E2 -16267.39} C_VEL
LIN {X 0,Y 304.4,Z 555.705,A -85,B 0,C 180,E1 -16269.384,E2 -16269.384} C_VEL
LIN {X 0,Y 302.626,Z 564.001,A -85,B 0,C 180,E1 -16271.026,E2 -16271.026} C_VEL
LIN {X 0,Y 300.587,Z 572.518,A -85,B 0,C 180,E1 -16273.006,E2 -16273.006} C_VEL
LIN {X 0,Y 299.055,Z 579.723,A -85,B 0,C 180,E1 -16275.018,E2 -16275.018} C_VEL
LIN {X 0,Y 297.818,Z 587.501,A -85,B 0,C 180,E1 -16277.738,E2 -16277.738} C_VEL
LIN {X 0,Y 297.335,Z 592.862,A -85,B 0,C 180,E1 -16279.789,E2 -16279.789} C_VEL
LIN {X 0,Y 297.284,Z 597.093,A -85,B 0,C 180,E1 -16281.845,E2 -16281.845} C_VEL
LIN {X 0,Y 297.391,Z 599.305,A -85,B 0,C 180,E1 -16283.214,E2 -16283.214} C_VEL
LIN {X 0,Y 297.571,Z 601.086,A -85,B 0,C 180,E1 -16284.579,E2 -16284.579} C_VEL
LIN {X 0,Y 297.844,Z 602.459,A -85,B 0,C 180,E1 -16285.94,E2 -16285.94} C_VEL
LIN {X 0,Y 297.938,Z 603.378,A -85,B 0,C 180,E1 -16287.296,E2 -16287.296} C_VEL
LIN {X 0,Y 298.359,Z 603.893,A -85,B 0,C 180,E1 -16288.65,E2 -16288.65} C_VEL
LIN {X 0,Y 298.591,Z 603.975,A -85,B 0,C 180,E1 -16290,E2 -16290} C_VEL
LIN {X 0,Y 298.382,Z 603.588,A -85,B 0,C 180,E1 -16291.349,E2 -16291.349} C_VEL
LIN {X 0,Y 297.994,Z 602.756,A -85,B 0,C 180,E1 -16292.703,E2 -16292.703} C_VEL
LIN {X 0,Y 297.904,Z 601.502,A -85,B 0,C 180,E1 -16294.058,E2 -16294.058} C_VEL
LIN {X 0,Y 297.558,Z 598.786,A -85,B 0,C 180,E1 -16296.101,E2 -16296.101} C_VEL
LIN {X 0,Y 297.383,Z 595.024,A -85,B 0,C 180,E1 -16298.152,E2 -16298.152} C_VEL
LIN {X 0,Y 297.433,Z 590.125,A -85,B 0,C 180,E1 -16300.207,E2 -16300.207} C_VEL
LIN {X 0,Y 297.984,Z 582.817,A -85,B 0,C 180,E1 -16302.601,E2 -16302.601} C_VEL
LIN {X 0,Y 298.709,Z 574.918,A -85,B 0,C 180,E1 -16304.65,E2 -16304.65} C_VEL
LIN {X 0,Y 299.935,Z 566.924,A -85,B 0,C 180,E1 -16306.33,E2 -16306.33} C_VEL
LIN {X 0,Y 301.235,Z 557.156,A -85,B 0,C 180,E1 -16308.007,E2 -16308.007} C_VEL
LIN {X 0,Y 301.681,Z 551.386,A -85,B 0,C 180,E1 -16308.858,E2 -16308.858} C_VEL
LIN {X 0,Y 301.909,Z 540.424,A -85,B 0,C 180,E1 -16310.259,E2 -16310.259} C_VEL
LIN {X 0,Y 301.803,Z 528.692,A -85,B 0,C 180,E1 -16311.47,E2 -16311.47} C_VEL
LIN {X 0,Y 301.104,Z 515.26,A -85,B 0,C 180,E1 -16312.563,E2 -16312.563} C_VEL
LIN {X 0,Y 299.657,Z 502.258,A -85,B 0,C 180,E1 -16313.387,E2 -16313.387} C_VEL
LIN {X 0,Y 298.165,Z 491.789,A -85,B 0,C 180,E1 -16313.912,E2 -16313.912} C_VEL
LIN {X 0,Y 299.12,Z 481.464,A -85,B 0,C 180,E1 -16318.028,E2 -16318.028} C_VEL
LIN {X 0,Y 300.315,Z 472.069,A -85,B 0,C 180,E1 -16321.772,E2 -16321.772} C_VEL
LIN {X 0,Y 301.583,Z 462.538,A -85,B 0,C 180,E1 -16325.633,E2 -16325.633} C_VEL
LIN {X 0,Y 302.457,Z 457.21,A -85,B 0,C 180,E1 -16327.811,E2 -16327.811} C_VEL
LIN {X 0,Y 302.037,Z 452.59,A -85,B 0,C 180,E1 -16329.837,E2 -16329.837} C_VEL
LIN {X 0,Y 300.535,Z 444.662,A -85,B 0,C 180,E1 -16333.537,E2 -16333.537} C_VEL
LIN {X 0,Y 299.056,Z 437.639,A -85,B 0,C 180,E1 -16337.038,E2 -16337.038} C_VEL
LIN {X 0,Y 298.388,Z 434.321,A -85,B 0,C 180,E1 -16338.825,E2 -16338.825} C_VEL
LIN {X 0,Y 298.432,Z 434.312,A -85,B 0,C 180,E1 -16342.245,E2 -16342.245} C_VEL
LIN {X 0,Y 298.409,Z 434.314,A -85,B 0,C 180,E1 -16345.581,E2 -16345.581} C_VEL
LIN {X 0,Y 298.392,Z 434.316,A -85,B 0,C 180,E1 -16348.791,E2 -16348.791} C_VEL
LIN {X 0,Y 298.459,Z 434.309,A -85,B 0,C 180,E1 -16351.904,E2 -16351.904} C_VEL
LIN {X 0,Y 298.486,Z 434.302,A -85,B 0,C 180,E1 -16354.924,E2 -16354.924} C_VEL
LIN {X 0,Y 298.464,Z 434.306,A -85,B 0,C 180,E1 -16359.316,E2 -16359.316} C_VEL
LIN {X 0,Y 298.539,Z 434.301,A -85,B 0,C 180,E1 -16362.18,E2 -16362.18} C_VEL
LIN {X 0,Y 298.594,Z 434.289,A -85,B 0,C 180,E1 -16364.995,E2 -16364.995} C_VEL
LIN {X 0,Y 298.594,Z 434.289,A -85,B 0,C 180,E1 -16369.147,E2 -16369.147} C_VEL
LIN {X 0,Y 298.719,Z 434.277,A -85,B 0,C 180,E1 -16371.885,E2 -16371.885} C_VEL
LIN {X 0,Y 298.657,Z 434.281,A -85,B 0,C 180,E1 -16374.599,E2 -16374.599} C_VEL
LIN {X 0,Y 298.925,Z 434.248,A -85,B 0,C 180,E1 -16378.653,E2 -16378.653} C_VEL
LIN {X 0,Y 298.925,Z 434.247,A -85,B 0,C 180,E1 -16381.347,E2 -16381.347} C_VEL
LIN {X 0,Y 298.799,Z 434.26,A -85,B 0,C 180,E1 -16386.754,E2 -16386.754} C_VEL
LIN {X 0,Y 298.681,Z 434.278,A -85,B 0,C 180,E1 -16389.481,E2 -16389.481} C_VEL
LIN {X 0,Y 298.553,Z 434.291,A -85,B 0,C 180,E1 -16393.616,E2 -16393.616} C_VEL
LIN {X 0,Y 298.55,Z 434.295,A -85,B 0,C 180,E1 -16396.409,E2 -16396.409} C_VEL
LIN {X 0,Y 298.513,Z 434.298,A -85,B 0,C 180,E1 -16399.655,E2 -16399.655} C_VEL
LIN {X 0,Y 298.458,Z 434.296,A -85,B 0,C 180,E1 -16403.598,E2 -16403.598} C_VEL
LIN {X 0,Y 298.49,Z 434.301,A -85,B 0,C 180,E1 -16406.575,E2 -16406.575} C_VEL
LIN {X 0,Y 298.417,Z 434.313,A -85,B 0,C 180,E1 -16409.642,E2 -16409.642} C_VEL
LIN {X 0,Y 298.396,Z 434.303,A -85,B 0,C 180,E1 -16412.801,E2 -16412.801} C_VEL
LIN {X 0,Y 298.466,Z 434.304,A -85,B 0,C 180,E1 -16416.813,E2 -16416.813} C_VEL
LIN {X 0,Y 298.388,Z 434.312,A -85,B 0,C 180,E1 -16421.088,E2 -16421.088} C_VEL
LIN {X 0,Y 298.4,Z 434.312,A -85,B 0,C 180,E1 -16423.104,E2 -16423.104} C_VEL
LIN {X 0,Y 298.404,Z 434.31,A -85,B 0,C 180,E1 -16426.921,E2 -16426.921} C_VEL
LIN {X 0,Y 298.417,Z 434.308,A -85,B 0,C 180,E1 -16431.004,E2 -16431.004} C_VEL
LIN {X 0,Y 298.434,Z 434.309,A -85,B 0,C 180,E1 -16433.933,E2 -16433.933} C_VEL
LIN {X 0,Y 298.402,Z 434.315,A -85,B 0,C 180,E1 -16437.982,E2 -16437.982} C_VEL
LIN {X 0,Y 298.479,Z 434.303,A -85,B 0,C 180,E1 -16441.906,E2 -16441.906} C_VEL
LIN {X 0,Y 298.489,Z 434.3,A -85,B 0,C 180,E1 -16444.925,E2 -16444.925} C_VEL
LIN {X 0,Y 298.454,Z 434.309,A -85,B 0,C 180,E1 -16449.316,E2 -16449.316} C_VEL
LIN {X 0,Y 298.533,Z 434.4,A -85,B 0,C 180,E1 -16450.273,E2 -16450.273} C_VEL
LIN {X 0,Y 302.683,Z 446.095,A -85,B 0,C 180,E1 -16451.567,E2 -16451.567} C_VEL
LIN {X 0,Y 305.892,Z 456.917,A -85,B 0,C 180,E1 -16452.966,E2 -16452.966} C_VEL
LIN {X 0,Y 306.875,Z 460.866,A -85,B 0,C 180,E1 -16453.536,E2 -16453.536} C_VEL
LIN {X 0,Y 305.907,Z 470.639,A -85,B 0,C 180,E1 -16454.852,E2 -16454.852} C_VEL
LIN {X 0,Y 304.615,Z 479.898,A -85,B 0,C 180,E1 -16456.368,E2 -16456.368} C_VEL
LIN {X 0,Y 303.35,Z 487.891,A -85,B 0,C 180,E1 -16457.965,E2 -16457.965} C_VEL
LIN {X 0,Y 302.119,Z 495.908,A -85,B 0,C 180,E1 -16459.953,E2 -16459.953} C_VEL
LIN {X 0,Y 301.032,Z 502.369,A -85,B 0,C 180,E1 -16461.948,E2 -16461.948} C_VEL
LIN {X 0,Y 300.333,Z 507.49,A -85,B 0,C 180,E1 -16463.956,E2 -16463.956} C_VEL
LIN {X 0,Y 299.537,Z 511.52,A -85,B 0,C 180,E1 -16465.964,E2 -16465.964} C_VEL
LIN {X 0,Y 299.152,Z 513.642,A -85,B 0,C 180,E1 -16467.307,E2 -16467.307} C_VEL
LIN {X 0,Y 298.8,Z 516.548,A -85,B 0,C 180,E1 -16470,E2 -16470} C_VEL
LIN {X 0,Y 298.784,Z 517.422,A -85,B 0,C 180,E1 -16471.348,E2 -16471.348} C_VEL
LIN {X 0,Y 298.669,Z 517.922,A -85,B 0,C 180,E1 -16472.698,E2 -16472.698} C_VEL
LIN {X 0,Y 298.573,Z 518.027,A -85,B 0,C 180,E1 -16474.05,E2 -16474.05} C_VEL
LIN {X 0,Y 299.106,Z 517.053,A -85,B 0,C 180,E1 -16476.747,E2 -16476.747} C_VEL
LIN {X 0,Y 299.573,Z 515.968,A -85,B 0,C 180,E1 -16478.092,E2 -16478.092} C_VEL
LIN {X 0,Y 300.36,Z 512.784,A -85,B 0,C 180,E1 -16480.658,E2 -16480.658} C_VEL
LIN {X 0,Y 301.336,Z 508.888,A -85,B 0,C 180,E1 -16482.801,E2 -16482.801} C_VEL
LIN {X 0,Y 302.257,Z 504.106,A -85,B 0,C 180,E1 -16484.82,E2 -16484.82} C_VEL
LIN {X 0,Y 303.47,Z 498.049,A -85,B 0,C 180,E1 -16486.827,E2 -16486.827} C_VEL
LIN {X 0,Y 304.986,Z 490.43,A -85,B 0,C 180,E1 -16488.821,E2 -16488.821} C_VEL
LIN {X 0,Y 306.438,Z 482.612,A -85,B 0,C 180,E1 -16490.472,E2 -16490.472} C_VEL
LIN {X 0,Y 307.844,Z 473.062,A -85,B 0,C 180,E1 -16492.129,E2 -16492.129} C_VEL
LIN {X 0,Y 308.819,Z 466.109,A -85,B 0,C 180,E1 -16493.13,E2 -16493.13} C_VEL
LIN {X 0,Y 308.775,Z 464.343,A -85,B 0,C 180,E1 -16493.383,E2 -16493.383} C_VEL
LIN {X 0,Y 306.133,Z 455.071,A -85,B 0,C 180,E1 -16494.82,E2 -16494.82} C_VEL
LIN {X 0,Y 302.764,Z 445.249,A -85,B 0,C 180,E1 -16496.171,E2 -16496.171} C_VEL
LIN {X 0,Y 298.536,Z 434.602,A -85,B 0,C 180,E1 -16497.463,E2 -16497.463} C_VEL
LIN {X 0,Y 298.478,Z 434.303,A -85,B 0,C 180,E1 -16497.549,E2 -16497.549} C_VEL
LIN {X 0,Y 298.4,Z 434.314,A -85,B 0,C 180,E1 -16501.209,E2 -16501.209} C_VEL
LIN {X 0,Y 298.432,Z 434.312,A -85,B 0,C 180,E1 -16504.487,E2 -16504.487} C_VEL
LIN {X 0,Y 298.435,Z 434.311,A -85,B 0,C 180,E1 -16507.756,E2 -16507.756} C_VEL
LIN {X 0,Y 298.388,Z 434.315,A -85,B 0,C 180,E1 -16511.262,E2 -16511.262} C_VEL
LIN {X 0,Y 298.357,Z 434.318,A -85,B 0,C 180,E1 -16515.035,E2 -16515.035} C_VEL
LIN {X 0,Y 298.388,Z 434.314,A -85,B 0,C 180,E1 -16518.738,E2 -16518.738} C_VEL
LIN {X 0,Y 298.435,Z 434.311,A -85,B 0,C 180,E1 -16522.244,E2 -16522.244} C_VEL
LIN {X 0,Y 298.412,Z 434.312,A -85,B 0,C 180,E1 -16525.581,E2 -16525.581} C_VEL
LIN {X 0,Y 298.399,Z 434.312,A -85,B 0,C 180,E1 -16528.791,E2 -16528.791} C_VEL
LIN {X 0,Y 298.467,Z 434.306,A -85,B 0,C 180,E1 -16531.904,E2 -16531.904} C_VEL
LIN {X 0,Y 298.488,Z 434.301,A -85,B 0,C 180,E1 -16534.924,E2 -16534.924} C_VEL
LIN {X 0,Y 298.444,Z 434.308,A -85,B 0,C 180,E1 -16539.315,E2 -16539.315} C_VEL
LIN {X 0,Y 298.605,Z 434.388,A -85,B 0,C 180,E1 -16541.762,E2 -16541.762} C_VEL
LIN {X 0,Y 301.407,Z 446.19,A -85,B 0,C 180,E1 -16542.944,E2 -16542.944} C_VEL
LIN {X 0,Y 302.8,Z 451.959,A -85,B 0,C 180,E1 -16543.613,E2 -16543.613} C_VEL
LIN {X 0,Y 301.955,Z 464.407,A -85,B 0,C 180,E1 -16545.165,E2 -16545.165} C_VEL
LIN {X 0,Y 301.251,Z 474.363,A -85,B 0,C 180,E1 -16546.68,E2 -16546.68} C_VEL
LIN {X 0,Y 300.381,Z 484.372,A -85,B 0,C 180,E1 -16548.529,E2 -16548.529} C_VEL
LIN {X 0,Y 299.716,Z 493.382,A -85,B 0,C 180,E1 -16550.552,E2 -16550.552} C_VEL
LIN {X 0,Y 299.242,Z 499.043,A -85,B 0,C 180,E1 -16552.081,E2 -16552.081} C_VEL
LIN {X 0,Y 298.423,Z 502.267,A -85,B 0,C 180,E1 -16553.016,E2 -16553.016} C_VEL
LIN {X 0,Y 295.257,Z 507.137,A -85,B 0,C 180,E1 -16554.569,E2 -16554.569} C_VEL
LIN {X 0,Y 292.158,Z 511.335,A -85,B 0,C 180,E1 -16556.221,E2 -16556.221} C_VEL
LIN {X 0,Y 291.467,Z 513.506,A -85,B 0,C 180,E1 -16557.294,E2 -16557.294} C_VEL
LIN {X 0,Y 291.585,Z 516.92,A -85,B 0,C 180,E1 -16559.309,E2 -16559.309} C_VEL
LIN {X 0,Y 291.834,Z 519.478,A -85,B 0,C 180,E1 -16561.38,E2 -16561.38} C_VEL
LIN {X 0,Y 292.377,Z 521.447,A -85,B 0,C 180,E1 -16564.135,E2 -16564.135} C_VEL
LIN {X 0,Y 292.823,Z 521.864,A -85,B 0,C 180,E1 -16565.509,E2 -16565.509} C_VEL
LIN {X 0,Y 293.393,Z 521.844,A -85,B 0,C 180,E1 -16566.879,E2 -16566.879} C_VEL
LIN {X 0,Y 294.94,Z 520.61,A -85,B 0,C 180,E1 -16569.602,E2 -16569.602} C_VEL
LIN {X 0,Y 295.857,Z 519.431,A -85,B 0,C 180,E1 -16570.955,E2 -16570.955} C_VEL
LIN {X 0,Y 297.446,Z 516.866,A -85,B 0,C 180,E1 -16572.971,E2 -16572.971} C_VEL
LIN {X 0,Y 299.291,Z 513.298,A -85,B 0,C 180,E1 -16574.969,E2 -16574.969} C_VEL
LIN {X 0,Y 301.806,Z 507.734,A -85,B 0,C 180,E1 -16577.302,E2 -16577.302} C_VEL
LIN {X 0,Y 304.252,Z 501.84,A -85,B 0,C 180,E1 -16579.218,E2 -16579.218} C_VEL
LIN {X 0,Y 306.953,Z 494.459,A -85,B 0,C 180,E1 -16581.138,E2 -16581.138} C_VEL
LIN {X 0,Y 309.956,Z 485.485,A -85,B 0,C 180,E1 -16583.025,E2 -16583.025} C_VEL
LIN {X 0,Y 311.936,Z 478.771,A -85,B 0,C 180,E1 -16584.195,E2 -16584.195} C_VEL
LIN {X 0,Y 310.622,Z 471.673,A -85,B 0,C 180,E1 -16586.056,E2 -16586.056} C_VEL
LIN {X 0,Y 308.881,Z 465.689,A -85,B 0,C 180,E1 -16587.711,E2 -16587.711} C_VEL
LIN {X 0,Y 306.674,Z 459.951,A -85,B 0,C 180,E1 -16589.443,E2 -16589.443} C_VEL
LIN {X 0,Y 303.077,Z 453.012,A -85,B 0,C 180,E1 -16591.965,E2 -16591.965} C_VEL
LIN {X 0,Y 300.88,Z 449.371,A -85,B 0,C 180,E1 -16593.543,E2 -16593.543} C_VEL
LIN {X 0,Y 299.22,Z 447.454,A -85,B 0,C 180,E1 -16594.707,E2 -16594.707} C_VEL
LIN {X 0,Y 297.009,Z 445.105,A -85,B 0,C 180,E1 -16596.435,E2 -16596.435} C_VEL
LIN {X 0,Y 294.285,Z 443.199,A -85,B 0,C 180,E1 -16599.026,E2 -16599.026} C_VEL
LIN {X 0,Y 294.008,Z 442.946,A -85,B 0,C 180,E1 -16599.518,E2 -16599.518} C_VEL
LIN {X 0,Y 293.935,Z 444.424,A -85,B 0,C 180,E1 -16602.165,E2 -16602.165} C_VEL
LIN {X 0,Y 293.778,Z 446.989,A -85,B 0,C 180,E1 -16604.887,E2 -16604.887} C_VEL
LIN {X 0,Y 295.316,Z 454.679,A -85,B 0,C 180,E1 -16608.763,E2 -16608.763} C_VEL
LIN {X 0,Y 296.121,Z 459.221,A -85,B 0,C 180,E1 -16610.926,E2 -16610.926} C_VEL
LIN {X 0,Y 296.08,Z 461.363,A -85,B 0,C 180,E1 -16611.891,E2 -16611.891} C_VEL
LIN {X 0,Y 295.474,Z 464.846,A -85,B 0,C 180,E1 -16613.327,E2 -16613.327} C_VEL
LIN {X 0,Y 295.911,Z 469.519,A -85,B 0,C 180,E1 -16614.206,E2 -16614.206} C_VEL
LIN {X 0,Y 297.417,Z 475.806,A -85,B 0,C 180,E1 -16615.634,E2 -16615.634} C_VEL
LIN {X 0,Y 298.333,Z 481.999,A -85,B 0,C 180,E1 -16616.752,E2 -16616.752} C_VEL
LIN {X 0,Y 298.873,Z 484.617,A -85,B 0,C 180,E1 -16617.258,E2 -16617.258} C_VEL
LIN {X 0,Y 300.606,Z 496.719,A -85,B 0,C 180,E1 -16619.313,E2 -16619.313} C_VEL
LIN {X 0,Y 301.9,Z 512.506,A -85,B 0,C 180,E1 -16621.764,E2 -16621.764} C_VEL
LIN {X 0,Y 301.927,Z 528.025,A -85,B 0,C 180,E1 -16624.122,E2 -16624.122} C_VEL
LIN {X 0,Y 301.016,Z 537.515,A -85,B 0,C 180,E1 -16625.583,E2 -16625.583} C_VEL
LIN {X 0,Y 298.747,Z 551.143,A -85,B 0,C 180,E1 -16627.889,E2 -16627.889} C_VEL
LIN {X 0,Y 296.776,Z 561.272,A -85,B 0,C 180,E1 -16629.917,E2 -16629.917} C_VEL
LIN {X 0,Y 294.08,Z 571.281,A -85,B 0,C 180,E1 -16632.259,E2 -16632.259} C_VEL
LIN {X 0,Y 292.123,Z 579.431,A -85,B 0,C 180,E1 -16634.654,E2 -16634.654} C_VEL
LIN {X 0,Y 291.047,Z 585.221,A -85,B 0,C 180,E1 -16636.738,E2 -16636.738} C_VEL
LIN {X 0,Y 290.226,Z 593.406,A -85,B 0,C 180,E1 -16640.24,E2 -16640.24} C_VEL
LIN {X 0,Y 290.262,Z 597.265,A -85,B 0,C 180,E1 -16642.348,E2 -16642.348} C_VEL
LIN {X 0,Y 290.481,Z 600.093,A -85,B 0,C 180,E1 -16644.446,E2 -16644.446} C_VEL
LIN {X 0,Y 290.77,Z 601.462,A -85,B 0,C 180,E1 -16645.841,E2 -16645.841} C_VEL
LIN {X 0,Y 290.89,Z 602.374,A -85,B 0,C 180,E1 -16647.23,E2 -16647.23} C_VEL
LIN {X 0,Y 291.322,Z 602.883,A -85,B 0,C 180,E1 -16648.617,E2 -16648.617} C_VEL
LIN {X 0,Y 291.576,Z 602.961,A -85,B 0,C 180,E1 -16650,E2 -16650} C_VEL
LIN {X 0,Y 291.319,Z 602.559,A -85,B 0,C 180,E1 -16651.382,E2 -16651.382} C_VEL
LIN {X 0,Y 290.946,Z 601.717,A -85,B 0,C 180,E1 -16652.769,E2 -16652.769} C_VEL
LIN {X 0,Y 290.854,Z 600.451,A -85,B 0,C 180,E1 -16654.157,E2 -16654.157} C_VEL
LIN {X 0,Y 290.483,Z 597.713,A -85,B 0,C 180,E1 -16656.25,E2 -16656.25} C_VEL
LIN {X 0,Y 290.307,Z 593.929,A -85,B 0,C 180,E1 -16658.352,E2 -16658.352} C_VEL
LIN {X 0,Y 290.394,Z 589.012,A -85,B 0,C 180,E1 -16660.458,E2 -16660.458} C_VEL
LIN {X 0,Y 290.989,Z 581.682,A -85,B 0,C 180,E1 -16662.909,E2 -16662.909} C_VEL
LIN {X 0,Y 291.717,Z 573.742,A -85,B 0,C 180,E1 -16665.01,E2 -16665.01} C_VEL
LIN {X 0,Y 293.092,Z 565.731,A -85,B 0,C 180,E1 -16666.723,E2 -16666.723} C_VEL
LIN {X 0,Y 294.433,Z 555.926,A -85,B 0,C 180,E1 -16668.437,E2 -16668.437} C_VEL
LIN {X 0,Y 294.87,Z 546.234,A -85,B 0,C 180,E1 -16669.855,E2 -16669.855} C_VEL
LIN {X 0,Y 295.001,Z 534.608,A -85,B 0,C 180,E1 -16671.256,E2 -16671.256} C_VEL
LIN {X 0,Y 294.689,Z 522.469,A -85,B 0,C 180,E1 -16672.431,E2 -16672.431} C_VEL
LIN {X 0,Y 293.774,Z 509.754,A -85,B 0,C 180,E1 -16673.401,E2 -16673.401} C_VEL
LIN {X 0,Y 292.045,Z 496.354,A -85,B 0,C 180,E1 -16674.19,E2 -16674.19} C_VEL
LIN {X 0,Y 291.164,Z 490.795,A -85,B 0,C 180,E1 -16674.463,E2 -16674.463} C_VEL
LIN {X 0,Y 292.224,Z 480.328,A -85,B 0,C 180,E1 -16678.751,E2 -16678.751} C_VEL
LIN {X 0,Y 293.463,Z 471.299,A -85,B 0,C 180,E1 -16682.459,E2 -16682.459} C_VEL
LIN {X 0,Y 294.926,Z 461.458,A -85,B 0,C 180,E1 -16686.565,E2 -16686.565} C_VEL
LIN {X 0,Y 295.503,Z 457.373,A -85,B 0,C 180,E1 -16688.294,E2 -16688.294} C_VEL
LIN {X 0,Y 294.9,Z 452.994,A -85,B 0,C 180,E1 -16690.304,E2 -16690.304} C_VEL
LIN {X 0,Y 293.392,Z 445.203,A -85,B 0,C 180,E1 -16694.059,E2 -16694.059} C_VEL
LIN {X 0,Y 291.695,Z 436.974,A -85,B 0,C 180,E1 -16698.323,E2 -16698.323} C_VEL
LIN {X 0,Y 291.346,Z 435.197,A -85,B 0,C 180,E1 -16699.36,E2 -16699.36} C_VEL
LIN {X 0,Y 291.425,Z 435.184,A -85,B 0,C 180,E1 -16702.922,E2 -16702.922} C_VEL
LIN {X 0,Y 291.345,Z 435.198,A -85,B 0,C 180,E1 -16706.302,E2 -16706.302} C_VEL
LIN {X 0,Y 291.383,Z 435.191,A -85,B 0,C 180,E1 -16710.261,E2 -16710.261} C_VEL
LIN {X 0,Y 291.415,Z 435.187,A -85,B 0,C 180,E1 -16714.272,E2 -16714.272} C_VEL
LIN {X 0,Y 291.39,Z 435.187,A -85,B 0,C 180,E1 -16717.3,E2 -16717.3} C_VEL
LIN {X 0,Y 291.463,Z 435.182,A -85,B 0,C 180,E1 -16720.271,E2 -16720.271} C_VEL
LIN {X 0,Y 291.555,Z 435.168,A -85,B 0,C 180,E1 -16724.624,E2 -16724.624} C_VEL
LIN {X 0,Y 291.538,Z 435.168,A -85,B 0,C 180,E1 -16728.881,E2 -16728.881} C_VEL
LIN {X 0,Y 291.669,Z 435.154,A -85,B 0,C 180,E1 -16731.688,E2 -16731.688} C_VEL
LIN {X 0,Y 291.627,Z 435.158,A -85,B 0,C 180,E1 -16734.468,E2 -16734.468} C_VEL
LIN {X 0,Y 291.891,Z 435.124,A -85,B 0,C 180,E1 -16738.621,E2 -16738.621} C_VEL
LIN {X 0,Y 291.891,Z 435.123,A -85,B 0,C 180,E1 -16741.38,E2 -16741.38} C_VEL
LIN {X 0,Y 291.748,Z 435.138,A -85,B 0,C 180,E1 -16746.918,E2 -16746.918} C_VEL
LIN {X 0,Y 291.63,Z 435.158,A -85,B 0,C 180,E1 -16749.712,E2 -16749.712} C_VEL
LIN {X 0,Y 291.523,Z 435.169,A -85,B 0,C 180,E1 -16753.951,E2 -16753.951} C_VEL
LIN {X 0,Y 291.488,Z 435.173,A -85,B 0,C 180,E1 -16756.818,E2 -16756.818} C_VEL
LIN {X 0,Y 291.451,Z 435.174,A -85,B 0,C 180,E1 -16759.875,E2 -16759.875} C_VEL
LIN {X 0,Y 291.401,Z 435.181,A -85,B 0,C 180,E1 -16764.206,E2 -16764.206} C_VEL
LIN {X 0,Y 291.422,Z 435.182,A -85,B 0,C 180,E1 -16767.272,E2 -16767.272} C_VEL
LIN {X 0,Y 291.335,Z 435.19,A -85,B 0,C 180,E1 -16770.437,E2 -16770.437} C_VEL
LIN {X 0,Y 291.346,Z 435.183,A -85,B 0,C 180,E1 -16773.699,E2 -16773.699} C_VEL
LIN {X 0,Y 291.395,Z 435.185,A -85,B 0,C 180,E1 -16777.259,E2 -16777.259} C_VEL
LIN {X 0,Y 291.335,Z 435.191,A -85,B 0,C 180,E1 -16780.643,E2 -16780.643} C_VEL
LIN {X 0,Y 291.291,Z 435.196,A -85,B 0,C 180,E1 -16784.402,E2 -16784.402} C_VEL
LIN {X 0,Y 291.328,Z 435.191,A -85,B 0,C 180,E1 -16788.405,E2 -16788.405} C_VEL
LIN {X 0,Y 291.366,Z 435.187,A -85,B 0,C 180,E1 -16791.161,E2 -16791.161} C_VEL
LIN {X 0,Y 291.387,Z 435.183,A -85,B 0,C 180,E1 -16794.63,E2 -16794.63} C_VEL
LIN {X 0,Y 291.378,Z 435.19,A -85,B 0,C 180,E1 -16797.952,E2 -16797.952} C_VEL
LIN {X 0,Y 291.393,Z 435.183,A -85,B 0,C 180,E1 -16801.16,E2 -16801.16} C_VEL
LIN {X 0,Y 291.424,Z 435.181,A -85,B 0,C 180,E1 -16804.273,E2 -16804.273} C_VEL
LIN {X 0,Y 291.385,Z 435.19,A -85,B 0,C 180,E1 -16807.3,E2 -16807.3} C_VEL
LIN {X 0,Y 291.479,Z 435.362,A -85,B 0,C 180,E1 -16809.718,E2 -16809.718} C_VEL
LIN {X 0,Y 295.896,Z 447.529,A -85,B 0,C 180,E1 -16811.121,E2 -16811.121} C_VEL
LIN {X 0,Y 299.077,Z 458.318,A -85,B 0,C 180,E1 -16812.566,E2 -16812.566} C_VEL
LIN {X 0,Y 300.2,Z 463.508,A -85,B 0,C 180,E1 -16813.335,E2 -16813.335} C_VEL
LIN {X 0,Y 298.797,Z 474.035,A -85,B 0,C 180,E1 -16814.831,E2 -16814.831} C_VEL
LIN {X 0,Y 297.302,Z 484.362,A -85,B 0,C 180,E1 -16816.675,E2 -16816.675} C_VEL
LIN {X 0,Y 295.861,Z 493.279,A -85,B 0,C 180,E1 -16818.699,E2 -16818.699} C_VEL
LIN {X 0,Y 294.581,Z 500.466,A -85,B 0,C 180,E1 -16820.733,E2 -16820.733} C_VEL
LIN {X 0,Y 293.625,Z 507.026,A -85,B 0,C 180,E1 -16823.127,E2 -16823.127} C_VEL
LIN {X 0,Y 292.802,Z 511.385,A -85,B 0,C 180,E1 -16825.181,E2 -16825.181} C_VEL
LIN {X 0,Y 292.137,Z 514.707,A -85,B 0,C 180,E1 -16827.242,E2 -16827.242} C_VEL
LIN {X 0,Y 291.774,Z 517.593,A -85,B 0,C 180,E1 -16830,E2 -16830} C_VEL
LIN {X 0,Y 291.761,Z 518.458,A -85,B 0,C 180,E1 -16831.381,E2 -16831.381} C_VEL
LIN {X 0,Y 291.646,Z 518.939,A -85,B 0,C 180,E1 -16832.763,E2 -16832.763} C_VEL
LIN {X 0,Y 291.555,Z 519.035,A -85,B 0,C 180,E1 -16834.147,E2 -16834.147} C_VEL
LIN {X 0,Y 292.124,Z 518.042,A -85,B 0,C 180,E1 -16836.909,E2 -16836.909} C_VEL
LIN {X 0,Y 292.612,Z 516.937,A -85,B 0,C 180,E1 -16838.286,E2 -16838.286} C_VEL
LIN {X 0,Y 293.455,Z 513.733,A -85,B 0,C 180,E1 -16840.911,E2 -16840.911} C_VEL
LIN {X 0,Y 294.48,Z 509.816,A -85,B 0,C 180,E1 -16843.105,E2 -16843.105} C_VEL
LIN {X 0,Y 295.448,Z 505.012,A -85,B 0,C 180,E1 -16845.169,E2 -16845.169} C_VEL
LIN {X 0,Y 296.731,Z 498.93,A -85,B 0,C 180,E1 -16847.221,E2 -16847.221} C_VEL
LIN {X 0,Y 298.328,Z 491.266,A -85,B 0,C 180,E1 -16849.258,E2 -16849.258} C_VEL
LIN {X 0,Y 299.849,Z 483.413,A -85,B 0,C 180,E1 -16850.943,E2 -16850.943} C_VEL
LIN {X 0,Y 301.323,Z 473.821,A -85,B 0,C 180,E1 -16852.634,E2 -16852.634} C_VEL
LIN {X 0,Y 302.262,Z 467.248,A -85,B 0,C 180,E1 -16853.6,E2 -16853.6} C_VEL
LIN {X 0,Y 299.849,Z 457.988,A -85,B 0,C 180,E1 -16855.102,E2 -16855.102} C_VEL
LIN {X 0,Y 296.553,Z 448.096,A -85,B 0,C 180,E1 -16856.537,E2 -16856.537} C_VEL
LIN {X 0,Y 292.632,Z 438.294,A -85,B 0,C 180,E1 -16857.815,E2 -16857.815} C_VEL
LIN {X 0,Y 291.473,Z 435.554,A -85,B 0,C 180,E1 -16858.148,E2 -16858.148} C_VEL
LIN {X 0,Y 291.417,Z 435.186,A -85,B 0,C 180,E1 -16858.191,E2 -16858.191} C_VEL
LIN {X 0,Y 291.349,Z 435.195,A -85,B 0,C 180,E1 -16862.404,E2 -16862.404} C_VEL
LIN {X 0,Y 291.389,Z 435.187,A -85,B 0,C 180,E1 -16865.371,E2 -16865.371} C_VEL
LIN {X 0,Y 291.368,Z 435.189,A -85,B 0,C 180,E1 -16868.84,E2 -16868.84} C_VEL
LIN {X 0,Y 291.323,Z 435.196,A -85,B 0,C 180,E1 -16872.492,E2 -16872.492} C_VEL
LIN {X 0,Y 291.313,Z 435.196,A -85,B 0,C 180,E1 -16876.366,E2 -16876.366} C_VEL
LIN {X 0,Y 291.391,Z 435.185,A -85,B 0,C 180,E1 -16880.517,E2 -16880.517} C_VEL
LIN {X 0,Y 291.428,Z 435.181,A -85,B 0,C 180,E1 -16882.922,E2 -16882.922} C_VEL
LIN {X 0,Y 291.349,Z 435.192,A -85,B 0,C 180,E1 -16886.302,E2 -16886.302} C_VEL
LIN {X 0,Y 291.391,Z 435.187,A -85,B 0,C 180,E1 -16890.26,E2 -16890.26} C_VEL
LIN {X 0,Y 291.42,Z 435.183,A -85,B 0,C 180,E1 -16894.272,E2 -16894.272} C_VEL
LIN {X 0,Y 291.378,Z 435.188,A -85,B 0,C 180,E1 -16897.299,E2 -16897.299} C_VEL
LIN {X 0,Y 291.531,Z 435.204,A -85,B 0,C 180,E1 -16901.554,E2 -16901.554} C_VEL
LIN {X 0,Y 294.325,Z 447.092,A -85,B 0,C 180,E1 -16902.774,E2 -16902.774} C_VEL
LIN {X 0,Y 295.764,Z 454.109,A -85,B 0,C 180,E1 -16903.61,E2 -16903.61} C_VEL
LIN {X 0,Y 294.862,Z 466.08,A -85,B 0,C 180,E1 -16905.154,E2 -16905.154} C_VEL
LIN {X 0,Y 294.217,Z 474.912,A -85,B 0,C 180,E1 -16906.532,E2 -16906.532} C_VEL
LIN {X 0,Y 293.27,Z 485.867,A -85,B 0,C 180,E1 -16908.597,E2 -16908.597} C_VEL
LIN {X 0,Y 292.587,Z 494.761,A -85,B 0,C 180,E1 -16910.669,E2 -16910.669} C_VEL
LIN {X 0,Y 291.954,Z 503.09,A -85,B 0,C 180,E1 -16913.087,E2 -16913.087} C_VEL
LIN {X 0,Y 291.544,Z 508.832,A -85,B 0,C 180,E1 -16915.16,E2 -16915.16} C_VEL
LIN {X 0,Y 291.467,Z 513.506,A -85,B 0,C 180,E1 -16917.294,E2 -16917.294} C_VEL
LIN {X 0,Y 290.857,Z 515.53,A -85,B 0,C 180,E1 -16918.382,E2 -16918.382} C_VEL
LIN {X 0,Y 288.154,Z 518.549,A -85,B 0,C 180,E1 -16920.174,E2 -16920.174} C_VEL
LIN {X 0,Y 285.939,Z 520.531,A -85,B 0,C 180,E1 -16921.651,E2 -16921.651} C_VEL
LIN {X 0,Y 285.112,Z 521.647,A -85,B 0,C 180,E1 -16922.809,E2 -16922.809} C_VEL
LIN {X 0,Y 285.112,Z 521.905,A -85,B 0,C 180,E1 -16923.202,E2 -16923.202} C_VEL
LIN {X 0,Y 285.854,Z 523.05,A -85,B 0,C 180,E1 -16925.644,E2 -16925.644} C_VEL
LIN {X 0,Y 286.468,Z 523.167,A -85,B 0,C 180,E1 -16927.046,E2 -16927.046} C_VEL
LIN {X 0,Y 287.224,Z 522.863,A -85,B 0,C 180,E1 -16928.442,E2 -16928.442} C_VEL
LIN {X 0,Y 289.1,Z 521.077,A -85,B 0,C 180,E1 -16931.214,E2 -16931.214} C_VEL
LIN {X 0,Y 290.145,Z 519.607,A -85,B 0,C 180,E1 -16932.592,E2 -16932.592} C_VEL
LIN {X 0,Y 292.756,Z 515.348,A -85,B 0,C 180,E1 -16935.312,E2 -16935.312} C_VEL
LIN {X 0,Y 294.99,Z 510.994,A -85,B 0,C 180,E1 -16937.326,E2 -16937.326} C_VEL
LIN {X 0,Y 297.977,Z 504.431,A -85,B 0,C 180,E1 -16939.639,E2 -16939.639} C_VEL
LIN {X 0,Y 300.859,Z 497.465,A -85,B 0,C 180,E1 -16941.587,E2 -16941.587} C_VEL
LIN {X 0,Y 303.425,Z 490.445,A -85,B 0,C 180,E1 -16943.188,E2 -16943.188} C_VEL
LIN {X 0,Y 306.139,Z 482.565,A -85,B 0,C 180,E1 -16944.683,E2 -16944.683} C_VEL
LIN {X 0,Y 306.299,Z 481.342,A -85,B 0,C 180,E1 -16944.946,E2 -16944.946} C_VEL
LIN {X 0,Y 305.099,Z 474.394,A -85,B 0,C 180,E1 -16946.915,E2 -16946.915} C_VEL
LIN {X 0,Y 302.997,Z 467.155,A -85,B 0,C 180,E1 -16949.15,E2 -16949.15} C_VEL
LIN {X 0,Y 300.041,Z 460.143,A -85,B 0,C 180,E1 -16951.71,E2 -16951.71} C_VEL
LIN {X 0,Y 298.104,Z 456.264,A -85,B 0,C 180,E1 -16953.385,E2 -16953.385} C_VEL
LIN {X 0,Y 296.501,Z 454.086,A -85,B 0,C 180,E1 -16954.672,E2 -16954.672} C_VEL
LIN {X 0,Y 294.214,Z 451.589,A -85,B 0,C 180,E1 -16956.668,E2 -16956.668} C_VEL
LIN {X 0,Y 291.662,Z 449.666,A -85,B 0,C 180,E1 -16959.548,E2 -16959.548} C_VEL
LIN {X 0,Y 290.323,Z 450.112,A -85,B 0,C 180,E1 -16961.371,E2 -16961.371} C_VEL
LIN {X 0,Y 289.478,Z 451.175,A -85,B 0,C 180,E1 -16963.252,E2 -16963.252} C_VEL
LIN {X 0,Y 289.144,Z 453.089,A -85,B 0,C 180,E1 -16965.179,E2 -16965.179} C_VEL
LIN {X 0,Y 289.411,Z 457.336,A -85,B 0,C 180,E1 -16967.786,E2 -16967.786} C_VEL
LIN {X 0,Y 290.571,Z 462.81,A -85,B 0,C 180,E1 -16970.287,E2 -16970.287} C_VEL
LIN {X 0,Y 291.751,Z 468.183,A -85,B 0,C 180,E1 -16972.084,E2 -16972.084} C_VEL
LIN {X 0,Y 292.082,Z 469.864,A -85,B 0,C 180,E1 -16972.564,E2 -16972.564} C_VEL
LIN {X 0,Y 292.586,Z 476.025,A -85,B 0,C 180,E1 -16973.845,E2 -16973.845} C_VEL
LIN {X 0,Y 293.464,Z 480.524,A -85,B 0,C 180,E1 -16974.916,E2 -16974.916} C_VEL
LIN {X 0,Y 294.116,Z 486.629,A -85,B 0,C 180,E1 -16976.11,E2 -16976.11} C_VEL
LIN {X 0,Y 295.268,Z 496.943,A -85,B 0,C 180,E1 -16978.021,E2 -16978.021} C_VEL
LIN {X 0,Y 296.079,Z 507.848,A -85,B 0,C 180,E1 -16979.889,E2 -16979.889} C_VEL
LIN {X 0,Y 296.256,Z 521.531,A -85,B 0,C 180,E1 -16982.129,E2 -16982.129} C_VEL
LIN {X 0,Y 295.488,Z 534.555,A -85,B 0,C 180,E1 -16984.274,E2 -16984.274} C_VEL
LIN {X 0,Y 292.995,Z 548.497,A -85,B 0,C 180,E1 -16986.685,E2 -16986.685} C_VEL
LIN {X 0,Y 290.889,Z 558.676,A -85,B 0,C 180,E1 -16988.752,E2 -16988.752} C_VEL
LIN {X 0,Y 288.413,Z 567.454,A -85,B 0,C 180,E1 -16990.794,E2 -16990.794} C_VEL
LIN {X 0,Y 285.966,Z 576.18,A -85,B 0,C 180,E1 -16993.264,E2 -16993.264} C_VEL
LIN {X 0,Y 284.398,Z 583.047,A -85,B 0,C 180,E1 -16995.693,E2 -16995.693} C_VEL
LIN {X 0,Y 283.177,Z 592.44,A -85,B 0,C 180,E1 -16999.995,E2 -16999.995} C_VEL
LIN {X 0,Y 283.182,Z 596.283,A -85,B 0,C 180,E1 -17002.154,E2 -17002.154} C_VEL
LIN {X 0,Y 283.393,Z 599.1,A -85,B 0,C 180,E1 -17004.307,E2 -17004.307} C_VEL
LIN {X 0,Y 283.681,Z 600.464,A -85,B 0,C 180,E1 -17005.737,E2 -17005.737} C_VEL
LIN {X 0,Y 283.839,Z 601.367,A -85,B 0,C 180,E1 -17007.161,E2 -17007.161} C_VEL
LIN {X 0,Y 284.257,Z 601.868,A -85,B 0,C 180,E1 -17008.583,E2 -17008.583} C_VEL
LIN {X 0,Y 284.559,Z 601.947,A -85,B 0,C 180,E1 -17010,E2 -17010} C_VEL
LIN {X 0,Y 284.257,Z 601.531,A -85,B 0,C 180,E1 -17011.416,E2 -17011.416} C_VEL
LIN {X 0,Y 283.898,Z 600.676,A -85,B 0,C 180,E1 -17012.838,E2 -17012.838} C_VEL
LIN {X 0,Y 283.78,Z 599.397,A -85,B 0,C 180,E1 -17014.261,E2 -17014.261} C_VEL
LIN {X 0,Y 283.408,Z 596.639,A -85,B 0,C 180,E1 -17016.407,E2 -17016.407} C_VEL
LIN {X 0,Y 283.243,Z 592.835,A -85,B 0,C 180,E1 -17018.561,E2 -17018.561} C_VEL
LIN {X 0,Y 283.366,Z 587.899,A -85,B 0,C 180,E1 -17020.72,E2 -17020.72} C_VEL
LIN {X 0,Y 283.977,Z 580.541,A -85,B 0,C 180,E1 -17023.233,E2 -17023.233} C_VEL
LIN {X 0,Y 284.772,Z 572.568,A -85,B 0,C 180,E1 -17025.385,E2 -17025.385} C_VEL
LIN {X 0,Y 286.222,Z 564.53,A -85,B 0,C 180,E1 -17027.136,E2 -17027.136} C_VEL
LIN {X 0,Y 287.607,Z 554.687,A -85,B 0,C 180,E1 -17028.891,E2 -17028.891} C_VEL
LIN {X 0,Y 287.999,Z 543.585,A -85,B 0,C 180,E1 -17030.535,E2 -17030.535} C_VEL
LIN {X 0,Y 288.091,Z 532.199,A -85,B 0,C 180,E1 -17031.904,E2 -17031.904} C_VEL
LIN {X 0,Y 287.71,Z 519.773,A -85,B 0,C 180,E1 -17033.1,E2 -17033.1} C_VEL
LIN {X 0,Y 286.649,Z 506.727,A -85,B 0,C 180,E1 -17034.097,E2 -17034.097} C_VEL
LIN {X 0,Y 284.753,Z 493.423,A -85,B 0,C 180,E1 -17034.881,E2 -17034.881} C_VEL
LIN {X 0,Y 284.197,Z 489.747,A -85,B 0,C 180,E1 -17035.055,E2 -17035.055} C_VEL
LIN {X 0,Y 285.352,Z 479.209,A -85,B 0,C 180,E1 -17039.51,E2 -17039.51} C_VEL
LIN {X 0,Y 286.725,Z 469.659,A -85,B 0,C 180,E1 -17043.552,E2 -17043.552} C_VEL
LIN {X 0,Y 288.268,Z 460.38,A -85,B 0,C 180,E1 -17047.553,E2 -17047.553} C_VEL
LIN {X 0,Y 288.425,Z 457.644,A -85,B 0,C 180,E1 -17048.763,E2 -17048.763} C_VEL
LIN {X 0,Y 287.262,Z 450.889,A -85,B 0,C 180,E1 -17052.009,E2 -17052.009} C_VEL
LIN {X 0,Y 285.91,Z 444.076,A -85,B 0,C 180,E1 -17055.467,E2 -17055.467} C_VEL
LIN {X 0,Y 284.33,Z 436.095,A -85,B 0,C 180,E1 -17059.807,E2 -17059.807} C_VEL
LIN {X 0,Y 284.35,Z 436.065,A -85,B 0,C 180,E1 -17063.617,E2 -17063.617} C_VEL
LIN {X 0,Y 284.308,Z 436.071,A -85,B 0,C 180,E1 -17067.19,E2 -17067.19} C_VEL
LIN {X 0,Y 284.355,Z 436.066,A -85,B 0,C 180,E1 -17070.376,E2 -17070.376} C_VEL
LIN {X 0,Y 284.376,Z 436.06,A -85,B 0,C 180,E1 -17073.587,E2 -17073.587} C_VEL
LIN {X 0,Y 284.369,Z 436.063,A -85,B 0,C 180,E1 -17076.707,E2 -17076.707} C_VEL
LIN {X 0,Y 284.406,Z 436.058,A -85,B 0,C 180,E1 -17081.262,E2 -17081.262} C_VEL
LIN {X 0,Y 284.493,Z 436.049,A -85,B 0,C 180,E1 -17084.459,E2 -17084.459} C_VEL
LIN {X 0,Y 284.49,Z 436.048,A -85,B 0,C 180,E1 -17088.602,E2 -17088.602} C_VEL
LIN {X 0,Y 284.623,Z 436.03,A -85,B 0,C 180,E1 -17091.48,E2 -17091.48} C_VEL
LIN {X 0,Y 284.596,Z 436.035,A -85,B 0,C 180,E1 -17094.331,E2 -17094.331} C_VEL
LIN {X 0,Y 284.857,Z 436.001,A -85,B 0,C 180,E1 -17098.586,E2 -17098.586} C_VEL
LIN {X 0,Y 284.857,Z 435.999,A -85,B 0,C 180,E1 -17101.414,E2 -17101.414} C_VEL
LIN {X 0,Y 284.7,Z 436.016,A -85,B 0,C 180,E1 -17107.09,E2 -17107.09} C_VEL
LIN {X 0,Y 284.567,Z 436.04,A -85,B 0,C 180,E1 -17109.956,E2 -17109.956} C_VEL
LIN {X 0,Y 284.483,Z 436.047,A -85,B 0,C 180,E1 -17114.303,E2 -17114.303} C_VEL
LIN {X 0,Y 284.426,Z 436.053,A -85,B 0,C 180,E1 -17117.249,E2 -17117.249} C_VEL
LIN {X 0,Y 284.38,Z 436.05,A -85,B 0,C 180,E1 -17120.242,E2 -17120.242} C_VEL
LIN {X 0,Y 284.37,Z 436.051,A -85,B 0,C 180,E1 -17123.876,E2 -17123.876} C_VEL
LIN {X 0,Y 284.397,Z 436.056,A -85,B 0,C 180,E1 -17127.174,E2 -17127.174} C_VEL
LIN {X 0,Y 284.295,Z 436.066,A -85,B 0,C 180,E1 -17131.275,E2 -17131.275} C_VEL
LIN {X 0,Y 284.363,Z 436.057,A -85,B 0,C 180,E1 -17135.354,E2 -17135.354} C_VEL
LIN {X 0,Y 284.324,Z 436.068,A -85,B 0,C 180,E1 -17138.168,E2 -17138.168} C_VEL
LIN {X 0,Y 284.271,Z 436.074,A -85,B 0,C 180,E1 -17142.125,E2 -17142.125} C_VEL
LIN {X 0,Y 284.257,Z 436.074,A -85,B 0,C 180,E1 -17146.19,E2 -17146.19} C_VEL
LIN {X 0,Y 284.309,Z 436.068,A -85,B 0,C 180,E1 -17150.024,E2 -17150.024} C_VEL
LIN {X 0,Y 284.352,Z 436.064,A -85,B 0,C 180,E1 -17153.617,E2 -17153.617} C_VEL
LIN {X 0,Y 284.311,Z 436.067,A -85,B 0,C 180,E1 -17157.189,E2 -17157.189} C_VEL
LIN {X 0,Y 284.365,Z 436.058,A -85,B 0,C 180,E1 -17160.377,E2 -17160.377} C_VEL
LIN {X 0,Y 284.384,Z 436.063,A -85,B 0,C 180,E1 -17163.587,E2 -17163.587} C_VEL
LIN {X 0,Y 284.369,Z 436.062,A -85,B 0,C 180,E1 -17166.708,E2 -17166.708} C_VEL
LIN {X 0,Y 284.356,Z 436.065,A -85,B 0,C 180,E1 -17169.098,E2 -17169.098} C_VEL
LIN {X 0,Y 288.572,Z 447.346,A -85,B 0,C 180,E1 -17170.447,E2 -17170.447} C_VEL
LIN {X 0,Y 291.899,Z 458.299,A -85,B 0,C 180,E1 -17171.942,E2 -17171.942} C_VEL
LIN {X 0,Y 293.515,Z 464.819,A -85,B 0,C 180,E1 -17172.944,E2 -17172.944} C_VEL
LIN {X 0,Y 292.067,Z 475.293,A -85,B 0,C 180,E1 -17174.473,E2 -17174.473} C_VEL
LIN {X 0,Y 290.491,Z 485.572,A -85,B 0,C 180,E1 -17176.356,E2 -17176.356} C_VEL
LIN {X 0,Y 288.991,Z 494.449,A -85,B 0,C 180,E1 -17178.426,E2 -17178.426} C_VEL
LIN {X 0,Y 287.664,Z 501.608,A -85,B 0,C 180,E1 -17180.508,E2 -17180.508} C_VEL
LIN {X 0,Y 286.665,Z 508.131,A -85,B 0,C 180,E1 -17182.959,E2 -17182.959} C_VEL
LIN {X 0,Y 285.807,Z 512.469,A -85,B 0,C 180,E1 -17185.063,E2 -17185.063} C_VEL
LIN {X 0,Y 285.122,Z 515.771,A -85,B 0,C 180,E1 -17187.175,E2 -17187.175} C_VEL
LIN {X 0,Y 284.749,Z 518.638,A -85,B 0,C 180,E1 -17190,E2 -17190} C_VEL
LIN {X 0,Y 284.737,Z 519.492,A -85,B 0,C 180,E1 -17191.415,E2 -17191.415} C_VEL
LIN {X 0,Y 284.623,Z 519.956,A -85,B 0,C 180,E1 -17192.831,E2 -17192.831} C_VEL
LIN {X 0,Y 284.539,Z 520.043,A -85,B 0,C 180,E1 -17194.25,E2 -17194.25} C_VEL
LIN {X 0,Y 285.144,Z 519.03,A -85,B 0,C 180,E1 -17197.079,E2 -17197.079} C_VEL
LIN {X 0,Y 285.655,Z 517.906,A -85,B 0,C 180,E1 -17198.489,E2 -17198.489} C_VEL
LIN {X 0,Y 286.604,Z 514.608,A -85,B 0,C 180,E1 -17201.224,E2 -17201.224} C_VEL
LIN {X 0,Y 287.633,Z 510.744,A -85,B 0,C 180,E1 -17203.422,E2 -17203.422} C_VEL
LIN {X 0,Y 288.657,Z 505.919,A -85,B 0,C 180,E1 -17205.535,E2 -17205.535} C_VEL
LIN {X 0,Y 290.009,Z 499.809,A -85,B 0,C 180,E1 -17207.634,E2 -17207.634} C_VEL
LIN {X 0,Y 291.687,Z 492.104,A -85,B 0,C 180,E1 -17209.714,E2 -17209.714} C_VEL
LIN {X 0,Y 293.272,Z 484.216,A -85,B 0,C 180,E1 -17211.436,E2 -17211.436} C_VEL
LIN {X 0,Y 294.819,Z 474.582,A -85,B 0,C 180,E1 -17213.162,E2 -17213.162} C_VEL
LIN {X 0,Y 295.656,Z 468.842,A -85,B 0,C 180,E1 -17214.03,E2 -17214.03} C_VEL
LIN {X 0,Y 292.895,Z 458.798,A -85,B 0,C 180,E1 -17215.727,E2 -17215.727} C_VEL
LIN {X 0,Y 289.399,Z 448.489,A -85,B 0,C 180,E1 -17217.269,E2 -17217.269} C_VEL
LIN {X 0,Y 285.501,Z 439.128,A -85,B 0,C 180,E1 -17218.543,E2 -17218.543} C_VEL
LIN {X 0,Y 284.339,Z 436.066,A -85,B 0,C 180,E1 -17218.913,E2 -17218.913} C_VEL
LIN {X 0,Y 284.31,Z 436.07,A -85,B 0,C 180,E1 -17222.945,E2 -17222.945} C_VEL
LIN {X 0,Y 284.354,Z 436.066,A -85,B 0,C 180,E1 -17226.383,E2 -17226.383} C_VEL
LIN {X 0,Y 284.31,Z 436.072,A -85,B 0,C 180,E1 -17229.995,E2 -17229.995} C_VEL
LIN {X 0,Y 284.249,Z 436.077,A -85,B 0,C 180,E1 -17234.19,E2 -17234.19} C_VEL
LIN {X 0,Y 284.276,Z 436.075,A -85,B 0,C 180,E1 -17238.124,E2 -17238.124} C_VEL
LIN {X 0,Y 284.338,Z 436.067,A -85,B 0,C 180,E1 -17242.275,E2 -17242.275} C_VEL
LIN {X 0,Y 284.327,Z 436.065,A -85,B 0,C 180,E1 -17245.353,E2 -17245.353} C_VEL
LIN {X 0,Y 284.3,Z 436.068,A -85,B 0,C 180,E1 -17248.726,E2 -17248.726} C_VEL
LIN {X 0,Y 284.401,Z 436.056,A -85,B 0,C 180,E1 -17252.826,E2 -17252.826} C_VEL
LIN {X 0,Y 284.337,Z 436.064,A -85,B 0,C 180,E1 -17256.704,E2 -17256.704} C_VEL
LIN {X 0,Y 284.497,Z 436.088,A -85,B 0,C 180,E1 -17261.361,E2 -17261.361} C_VEL
LIN {X 0,Y 287.574,Z 449.225,A -85,B 0,C 180,E1 -17262.745,E2 -17262.745} C_VEL
LIN {X 0,Y 288.719,Z 454.404,A -85,B 0,C 180,E1 -17263.38,E2 -17263.38} C_VEL
LIN {X 0,Y 287.847,Z 466.427,A -85,B 0,C 180,E1 -17264.964,E2 -17264.964} C_VEL
LIN {X 0,Y 287.07,Z 476.355,A -85,B 0,C 180,E1 -17266.551,E2 -17266.551} C_VEL
LIN {X 0,Y 286.147,Z 487.195,A -85,B 0,C 180,E1 -17268.668,E2 -17268.668} C_VEL
LIN {X 0,Y 285.455,Z 496.056,A -85,B 0,C 180,E1 -17270.791,E2 -17270.791} C_VEL
LIN {X 0,Y 284.857,Z 504.386,A -85,B 0,C 180,E1 -17273.27,E2 -17273.27} C_VEL
LIN {X 0,Y 284.251,Z 510.937,A -85,B 0,C 180,E1 -17275.746,E2 -17275.746} C_VEL
LIN {X 0,Y 284.461,Z 515.29,A -85,B 0,C 180,E1 -17277.876,E2 -17277.876} C_VEL
LIN {X 0,Y 284.672,Z 518.626,A -85,B 0,C 180,E1 -17280,E2 -17280} C_VEL
LIN {X 0,Y 285.037,Z 521.671,A -85,B 0,C 180,E1 -17282.826,E2 -17282.826} C_VEL
LIN {X 0,Y 285.112,Z 521.905,A -85,B 0,C 180,E1 -17283.202,E2 -17283.202} C_VEL
LIN {X 0,Y 284.762,Z 522.733,A -85,B 0,C 180,E1 -17284.379,E2 -17284.379} C_VEL
LIN {X 0,Y 282.644,Z 523.786,A -85,B 0,C 180,E1 -17286.325,E2 -17286.325} C_VEL
LIN {X 0,Y 281.035,Z 524.199,A -85,B 0,C 180,E1 -17287.902,E2 -17287.902} C_VEL
LIN {X 0,Y 280.728,Z 524.108,A -85,B 0,C 180,E1 -17289.104,E2 -17289.104} C_VEL
LIN {X 0,Y 280.91,Z 523.929,A -85,B 0,C 180,E1 -17289.502,E2 -17289.502} C_VEL
LIN {X 0,Y 282.337,Z 522.718,A -85,B 0,C 180,E1 -17291.486,E2 -17291.486} C_VEL
LIN {X 0,Y 283.457,Z 521.388,A -85,B 0,C 180,E1 -17292.894,E2 -17292.894} C_VEL
LIN {X 0,Y 285.505,Z 518.565,A -85,B 0,C 180,E1 -17294.979,E2 -17294.979} C_VEL
LIN {X 0,Y 287.766,Z 514.761,A -85,B 0,C 180,E1 -17297.042,E2 -17297.042} C_VEL
LIN {X 0,Y 290.699,Z 509.238,A -85,B 0,C 180,E1 -17299.342,E2 -17299.342} C_VEL
LIN {X 0,Y 294.228,Z 501.652,A -85,B 0,C 180,E1 -17301.73,E2 -17301.73} C_VEL
LIN {X 0,Y 297.482,Z 493.827,A -85,B 0,C 180,E1 -17303.68,E2 -17303.68} C_VEL
LIN {X 0,Y 300.591,Z 485.548,A -85,B 0,C 180,E1 -17305.34,E2 -17305.34} C_VEL
LIN {X 0,Y 300.476,Z 481.855,A -85,B 0,C 180,E1 -17306.385,E2 -17306.385} C_VEL
LIN {X 0,Y 299.177,Z 474.994,A -85,B 0,C 180,E1 -17308.56,E2 -17308.56} C_VEL
LIN {X 0,Y 297.326,Z 469.009,A -85,B 0,C 180,E1 -17310.713,E2 -17310.713} C_VEL
LIN {X 0,Y 294.723,Z 462.717,A -85,B 0,C 180,E1 -17313.423,E2 -17313.423} C_VEL
LIN {X 0,Y 292.899,Z 459.946,A -85,B 0,C 180,E1 -17315.161,E2 -17315.161} C_VEL
LIN {X 0,Y 290.973,Z 457.834,A -85,B 0,C 180,E1 -17317.149,E2 -17317.149} C_VEL
LIN {X 0,Y 289.406,Z 456.589,A -85,B 0,C 180,E1 -17319.153,E2 -17319.153} C_VEL
LIN {X 0,Y 288.062,Z 456.768,A -85,B 0,C 180,E1 -17321.203,E2 -17321.203} C_VEL
LIN {X 0,Y 287.129,Z 457.995,A -85,B 0,C 180,E1 -17323.263,E2 -17323.263} C_VEL
LIN {X 0,Y 286.846,Z 459.408,A -85,B 0,C 180,E1 -17324.722,E2 -17324.722} C_VEL
LIN {X 0,Y 286.873,Z 463.502,A -85,B 0,C 180,E1 -17327.304,E2 -17327.304} C_VEL
LIN {X 0,Y 287.853,Z 469.444,A -85,B 0,C 180,E1 -17330.059,E2 -17330.059} C_VEL
LIN {X 0,Y 288.651,Z 474.908,A -85,B 0,C 180,E1 -17331.817,E2 -17331.817} C_VEL
LIN {X 0,Y 288.745,Z 479.839,A -85,B 0,C 180,E1 -17332.898,E2 -17332.898} C_VEL
LIN {X 0,Y 289.398,Z 484.491,A -85,B 0,C 180,E1 -17334.056,E2 -17334.056} C_VEL
LIN {X 0,Y 290.423,Z 499.375,A -85,B 0,C 180,E1 -17337.078,E2 -17337.078} C_VEL
LIN {X 0,Y 290.787,Z 512.616,A -85,B 0,C 180,E1 -17339.499,E2 -17339.499} C_VEL
LIN {X 0,Y 290.46,Z 524.174,A -85,B 0,C 180,E1 -17341.523,E2 -17341.523} C_VEL
LIN {X 0,Y 289.339,Z 536.38,A -85,B 0,C 180,E1 -17343.686,E2 -17343.686} C_VEL
LIN {X 0,Y 286.995,Z 547.876,A -85,B 0,C 180,E1 -17345.784,E2 -17345.784} C_VEL
LIN {X 0,Y 284.284,Z 559.318,A -85,B 0,C 180,E1 -17348.233,E2 -17348.233} C_VEL
LIN {X 0,Y 281.714,Z 567.703,A -85,B 0,C 180,E1 -17350.318,E2 -17350.318} C_VEL
LIN {X 0,Y 279.07,Z 576.304,A -85,B 0,C 180,E1 -17352.922,E2 -17352.922} C_VEL
LIN {X 0,Y 277.481,Z 582.644,A -85,B 0,C 180,E1 -17355.328,E2 -17355.328} C_VEL
LIN {X 0,Y 276.58,Z 587.322,A -85,B 0,C 180,E1 -17357.526,E2 -17357.526} C_VEL
LIN {X 0,Y 276.079,Z 594.158,A -85,B 0,C 180,E1 -17361.214,E2 -17361.214} C_VEL
LIN {X 0,Y 276.208,Z 596.632,A -85,B 0,C 180,E1 -17362.904,E2 -17362.904} C_VEL
LIN {X 0,Y 276.595,Z 599.466,A -85,B 0,C 180,E1 -17365.628,E2 -17365.628} C_VEL
LIN {X 0,Y 276.784,Z 600.361,A -85,B 0,C 180,E1 -17367.089,E2 -17367.089} C_VEL
LIN {X 0,Y 277.193,Z 600.854,A -85,B 0,C 180,E1 -17368.547,E2 -17368.547} C_VEL
LIN {X 0,Y 277.539,Z 600.932,A -85,B 0,C 180,E1 -17370,E2 -17370} C_VEL
LIN {X 0,Y 277.196,Z 600.503,A -85,B 0,C 180,E1 -17371.453,E2 -17371.453} C_VEL
LIN {X 0,Y 276.847,Z 599.634,A -85,B 0,C 180,E1 -17372.91,E2 -17372.91} C_VEL
LIN {X 0,Y 276.708,Z 598.342,A -85,B 0,C 180,E1 -17374.37,E2 -17374.37} C_VEL
LIN {X 0,Y 276.302,Z 594.523,A -85,B 0,C 180,E1 -17377.25,E2 -17377.25} C_VEL
LIN {X 0,Y 276.192,Z 590.237,A -85,B 0,C 180,E1 -17379.52,E2 -17379.52} C_VEL
LIN {X 0,Y 276.556,Z 583.842,A -85,B 0,C 180,E1 -17382.102,E2 -17382.102} C_VEL
LIN {X 0,Y 277.261,Z 576.907,A -85,B 0,C 180,E1 -17384.308,E2 -17384.308} C_VEL
LIN {X 0,Y 278.199,Z 569.889,A -85,B 0,C 180,E1 -17386.134,E2 -17386.134} C_VEL
LIN {X 0,Y 279.607,Z 561.498,A -85,B 0,C 180,E1 -17387.933,E2 -17387.933} C_VEL
LIN {X 0,Y 280.699,Z 553.428,A -85,B 0,C 180,E1 -17389.375,E2 -17389.375} C_VEL
LIN {X 0,Y 281.133,Z 542.277,A -85,B 0,C 180,E1 -17391.061,E2 -17391.061} C_VEL
LIN {X 0,Y 281.245,Z 530.712,A -85,B 0,C 180,E1 -17392.474,E2 -17392.474} C_VEL
LIN {X 0,Y 280.785,Z 517.588,A -85,B 0,C 180,E1 -17393.758,E2 -17393.758} C_VEL
LIN {X 0,Y 279.6,Z 504.576,A -85,B 0,C 180,E1 -17394.77,E2 -17394.77} C_VEL
LIN {X 0,Y 277.568,Z 491.193,A -85,B 0,C 180,E1 -17395.564,E2 -17395.564} C_VEL
LIN {X 0,Y 277.274,Z 488.64,A -85,B 0,C 180,E1 -17395.725,E2 -17395.725} C_VEL
LIN {X 0,Y 278.549,Z 478.094,A -85,B 0,C 180,E1 -17400.306,E2 -17400.306} C_VEL
LIN {X 0,Y 280.042,Z 468.369,A -85,B 0,C 180,E1 -17404.554,E2 -17404.554} C_VEL
LIN {X 0,Y 281.278,Z 461.188,A -85,B 0,C 180,E1 -17407.745,E2 -17407.745} C_VEL
LIN {X 0,Y 281.367,Z 457.93,A -85,B 0,C 180,E1 -17409.257,E2 -17409.257} C_VEL
LIN {X 0,Y 279.862,Z 449.903,A -85,B 0,C 180,E1 -17413.259,E2 -17413.259} C_VEL
LIN {X 0,Y 278.441,Z 442.799,A -85,B 0,C 180,E1 -17417.052,E2 -17417.052} C_VEL
LIN {X 0,Y 277.266,Z 436.95,A -85,B 0,C 180,E1 -17420.434,E2 -17420.434} C_VEL
LIN {X 0,Y 277.304,Z 436.945,A -85,B 0,C 180,E1 -17424.344,E2 -17424.344} C_VEL
LIN {X 0,Y 277.244,Z 436.952,A -85,B 0,C 180,E1 -17427.836,E2 -17427.836} C_VEL
LIN {X 0,Y 277.268,Z 436.946,A -85,B 0,C 180,E1 -17431.21,E2 -17431.21} C_VEL
LIN {X 0,Y 277.313,Z 436.942,A -85,B 0,C 180,E1 -17434.48,E2 -17434.48} C_VEL
LIN {X 0,Y 277.292,Z 436.944,A -85,B 0,C 180,E1 -17437.656,E2 -17437.656} C_VEL
LIN {X 0,Y 277.347,Z 436.938,A -85,B 0,C 180,E1 -17440.766,E2 -17440.766} C_VEL
LIN {X 0,Y 277.436,Z 436.926,A -85,B 0,C 180,E1 -17445.326,E2 -17445.326} C_VEL
LIN {X 0,Y 277.461,Z 436.924,A -85,B 0,C 180,E1 -17449.787,E2 -17449.787} C_VEL
LIN {X 0,Y 277.63,Z 436.901,A -85,B 0,C 180,E1 -17452.729,E2 -17452.729} C_VEL
LIN {X 0,Y 277.823,Z 436.877,A -85,B 0,C 180,E1 -17458.551,E2 -17458.551} C_VEL
LIN {X 0,Y 277.823,Z 436.876,A -85,B 0,C 180,E1 -17461.45,E2 -17461.45} C_VEL
LIN {X 0,Y 277.655,Z 436.893,A -85,B 0,C 180,E1 -17467.271,E2 -17467.271} C_VEL
LIN {X 0,Y 277.508,Z 436.917,A -85,B 0,C 180,E1 -17470.212,E2 -17470.212} C_VEL
LIN {X 0,Y 277.436,Z 436.923,A -85,B 0,C 180,E1 -17474.674,E2 -17474.674} C_VEL
LIN {X 0,Y 277.346,Z 436.931,A -85,B 0,C 180,E1 -17479.234,E2 -17479.234} C_VEL
LIN {X 0,Y 277.32,Z 436.931,A -85,B 0,C 180,E1 -17484.171,E2 -17484.171} C_VEL
LIN {X 0,Y 277.326,Z 436.939,A -85,B 0,C 180,E1 -17487.505,E2 -17487.505} C_VEL
LIN {X 0,Y 277.273,Z 436.94,A -85,B 0,C 180,E1 -17490.482,E2 -17490.482} C_VEL
LIN {X 0,Y 277.255,Z 436.936,A -85,B 0,C 180,E1 -17493.895,E2 -17493.895} C_VEL
LIN {X 0,Y 277.282,Z 436.944,A -85,B 0,C 180,E1 -17497.468,E2 -17497.468} C_VEL
LIN {X 0,Y 277.211,Z 436.951,A -85,B 0,C 180,E1 -17501.237,E2 -17501.237} C_VEL
LIN {X 0,Y 277.202,Z 436.95,A -85,B 0,C 180,E1 -17505.227,E2 -17505.227} C_VEL
LIN {X 0,Y 277.224,Z 436.949,A -85,B 0,C 180,E1 -17509.512,E2 -17509.512} C_VEL
LIN {X 0,Y 277.283,Z 436.941,A -85,B 0,C 180,E1 -17512.533,E2 -17512.533} C_VEL
LIN {X 0,Y 277.257,Z 436.947,A -85,B 0,C 180,E1 -17516.106,E2 -17516.106} C_VEL
LIN {X 0,Y 277.263,Z 436.948,A -85,B 0,C 180,E1 -17519.539,E2 -17519.539} C_VEL
LIN {X 0,Y 277.365,Z 436.933,A -85,B 0,C 180,E1 -17522.865,E2 -17522.865} C_VEL
LIN {X 0,Y 277.332,Z 436.938,A -85,B 0,C 180,E1 -17526.08,E2 -17526.08} C_VEL
LIN {X 0,Y 277.305,Z 437.077,A -85,B 0,C 180,E1 -17528.493,E2 -17528.493} C_VEL
LIN {X 0,Y 281.856,Z 449.047,A -85,B 0,C 180,E1 -17529.981,E2 -17529.981} C_VEL
LIN {X 0,Y 284.698,Z 458.278,A -85,B 0,C 180,E1 -17531.282,E2 -17531.282} C_VEL
LIN {X 0,Y 286.743,Z 466.188,A -85,B 0,C 180,E1 -17532.534,E2 -17532.534} C_VEL
LIN {X 0,Y 285.422,Z 476.029,A -85,B 0,C 180,E1 -17534.01,E2 -17534.01} C_VEL
LIN {X 0,Y 284.003,Z 485.057,A -85,B 0,C 180,E1 -17535.673,E2 -17535.673} C_VEL
LIN {X 0,Y 282.608,Z 492.89,A -85,B 0,C 180,E1 -17537.432,E2 -17537.432} C_VEL
LIN {X 0,Y 281.243,Z 500.556,A -85,B 0,C 180,E1 -17539.562,E2 -17539.562} C_VEL
LIN {X 0,Y 280.235,Z 505.753,A -85,B 0,C 180,E1 -17541.346,E2 -17541.346} C_VEL
LIN {X 0,Y 279.417,Z 510.806,A -85,B 0,C 180,E1 -17543.501,E2 -17543.501} C_VEL
LIN {X 0,Y 278.535,Z 514.773,A -85,B 0,C 180,E1 -17545.659,E2 -17545.659} C_VEL
LIN {X 0,Y 278.108,Z 516.834,A -85,B 0,C 180,E1 -17547.103,E2 -17547.103} C_VEL
LIN {X 0,Y 277.724,Z 519.682,A -85,B 0,C 180,E1 -17550,E2 -17550} C_VEL
LIN {X 0,Y 277.713,Z 520.524,A -85,B 0,C 180,E1 -17551.45,E2 -17551.45} C_VEL
LIN {X 0,Y 277.523,Z 521.051,A -85,B 0,C 180,E1 -17554.357,E2 -17554.357} C_VEL
LIN {X 0,Y 278.167,Z 520.017,A -85,B 0,C 180,E1 -17557.258,E2 -17557.258} C_VEL
LIN {X 0,Y 278.702,Z 518.875,A -85,B 0,C 180,E1 -17558.703,E2 -17558.703} C_VEL
LIN {X 0,Y 279.717,Z 515.552,A -85,B 0,C 180,E1 -17561.507,E2 -17561.507} C_VEL
LIN {X 0,Y 280.772,Z 511.675,A -85,B 0,C 180,E1 -17563.757,E2 -17563.757} C_VEL
LIN {X 0,Y 281.881,Z 506.825,A -85,B 0,C 180,E1 -17565.918,E2 -17565.918} C_VEL
LIN {X 0,Y 283.293,Z 500.687,A -85,B 0,C 180,E1 -17568.066,E2 -17568.066} C_VEL
LIN {X 0,Y 285.054,Z 492.943,A -85,B 0,C 180,E1 -17570.193,E2 -17570.193} C_VEL
LIN {X 0,Y 286.725,Z 485.019,A -85,B 0,C 180,E1 -17571.95,E2 -17571.95} C_VEL
LIN {X 0,Y 288.336,Z 475.344,A -85,B 0,C 180,E1 -17573.715,E2 -17573.715} C_VEL
LIN {X 0,Y 289.057,Z 470.804,A -85,B 0,C 180,E1 -17574.415,E2 -17574.415} C_VEL
LIN {X 0,Y 286.323,Z 460.578,A -85,B 0,C 180,E1 -17576.221,E2 -17576.221} C_VEL
LIN {X 0,Y 282.957,Z 450.756,A -85,B 0,C 180,E1 -17577.768,E2 -17577.768} C_VEL
LIN {X 0,Y 278.787,Z 440.68,A -85,B 0,C 180,E1 -17579.206,E2 -17579.206} C_VEL
LIN {X 0,Y 277.336,Z 436.939,A -85,B 0,C 180,E1 -17579.684,E2 -17579.684} C_VEL
LIN {X 0,Y 277.258,Z 436.95,A -85,B 0,C 180,E1 -17583.895,E2 -17583.895} C_VEL
LIN {X 0,Y 277.285,Z 436.945,A -85,B 0,C 180,E1 -17587.467,E2 -17587.467} C_VEL
LIN {X 0,Y 277.213,Z 436.953,A -85,B 0,C 180,E1 -17591.236,E2 -17591.236} C_VEL
LIN {X 0,Y 277.205,Z 436.953,A -85,B 0,C 180,E1 -17595.226,E2 -17595.226} C_VEL
LIN {X 0,Y 277.226,Z 436.952,A -85,B 0,C 180,E1 -17599.512,E2 -17599.512} C_VEL
LIN {X 0,Y 277.285,Z 436.944,A -85,B 0,C 180,E1 -17602.533,E2 -17602.533} C_VEL
LIN {X 0,Y 277.258,Z 436.949,A -85,B 0,C 180,E1 -17606.105,E2 -17606.105} C_VEL
LIN {X 0,Y 277.265,Z 436.947,A -85,B 0,C 180,E1 -17609.539,E2 -17609.539} C_VEL
LIN {X 0,Y 277.363,Z 436.933,A -85,B 0,C 180,E1 -17612.864,E2 -17612.864} C_VEL
LIN {X 0,Y 277.301,Z 436.942,A -85,B 0,C 180,E1 -17616.077,E2 -17616.077} C_VEL
LIN {X 0,Y 277.458,Z 437.016,A -85,B 0,C 180,E1 -17621.182,E2 -17621.182} C_VEL
LIN {X 0,Y 280.236,Z 449.167,A -85,B 0,C 180,E1 -17622.485,E2 -17622.485} C_VEL
LIN {X 0,Y 281.644,Z 456.086,A -85,B 0,C 180,E1 -17623.348,E2 -17623.348} C_VEL
LIN {X 0,Y 280.726,Z 467.842,A -85,B 0,C 180,E1 -17624.945,E2 -17624.945} C_VEL
LIN {X 0,Y 279.946,Z 477.711,A -85,B 0,C 180,E1 -17626.572,E2 -17626.572} C_VEL
LIN {X 0,Y 279.035,Z 488.529,A -85,B 0,C 180,E1 -17628.744,E2 -17628.744} C_VEL
LIN {X 0,Y 278.342,Z 497.353,A -85,B 0,C 180,E1 -17630.92,E2 -17630.92} C_VEL
LIN {X 0,Y 277.816,Z 504.563,A -85,B 0,C 180,E1 -17633.098,E2 -17633.098} C_VEL
LIN {X 0,Y 277.194,Z 511.346,A -85,B 0,C 180,E1 -17635.637,E2 -17635.637} C_VEL
LIN {X 0,Y 277.388,Z 515.876,A -85,B 0,C 180,E1 -17637.822,E2 -17637.822} C_VEL
LIN {X 0,Y 277.621,Z 519.39,A -85,B 0,C 180,E1 -17640,E2 -17640} C_VEL
LIN {X 0,Y 278.025,Z 522.623,A -85,B 0,C 180,E1 -17642.898,E2 -17642.898} C_VEL
LIN {X 0,Y 278.388,Z 523.651,A -85,B 0,C 180,E1 -17644.343,E2 -17644.343} C_VEL
LIN {X 0,Y 279.539,Z 524.453,A -85,B 0,C 180,E1 -17647.221,E2 -17647.221} C_VEL
LIN {X 0,Y 280.91,Z 523.929,A -85,B 0,C 180,E1 -17649.502,E2 -17649.502} C_VEL
LIN {X 0,Y 281.11,Z 523.475,A -85,B 0,C 180,E1 -17650.702,E2 -17650.702} C_VEL
LIN {X 0,Y 279.89,Z 522.638,A -85,B 0,C 180,E1 -17652.703,E2 -17652.703} C_VEL
LIN {X 0,Y 278.975,Z 521.563,A -85,B 0,C 180,E1 -17654.303,E2 -17654.303} C_VEL
LIN {X 0,Y 279.161,Z 520.316,A -85,B 0,C 180,E1 -17655.485,E2 -17655.485} C_VEL
LIN {X 0,Y 279.498,Z 519.777,A -85,B 0,C 180,E1 -17655.867,E2 -17655.867} C_VEL
LIN {X 0,Y 282.194,Z 515.652,A -85,B 0,C 180,E1 -17658.138,E2 -17658.138} C_VEL
LIN {X 0,Y 285.585,Z 509.643,A -85,B 0,C 180,E1 -17660.566,E2 -17660.566} C_VEL
LIN {X 0,Y 288.708,Z 503.495,A -85,B 0,C 180,E1 -17662.544,E2 -17662.544} C_VEL
LIN {X 0,Y 292.184,Z 495.776,A -85,B 0,C 180,E1 -17664.514,E2 -17664.514} C_VEL
LIN {X 0,Y 295.139,Z 488.652,A -85,B 0,C 180,E1 -17666.017,E2 -17666.017} C_VEL
LIN {X 0,Y 295.168,Z 485.783,A -85,B 0,C 180,E1 -17666.897,E2 -17666.897} C_VEL
LIN {X 0,Y 294.163,Z 479.018,A -85,B 0,C 180,E1 -17669.223,E2 -17669.223} C_VEL
LIN {X 0,Y 292.858,Z 474.011,A -85,B 0,C 180,E1 -17671.18,E2 -17671.18} C_VEL
LIN {X 0,Y 290.911,Z 468.475,A -85,B 0,C 180,E1 -17673.755,E2 -17673.755} C_VEL
LIN {X 0,Y 290.232,Z 467.105,A -85,B 0,C 180,E1 -17674.581,E2 -17674.581} C_VEL
LIN {X 0,Y 288.506,Z 464.938,A -85,B 0,C 180,E1 -17676.497,E2 -17676.497} C_VEL
LIN {X 0,Y 287.063,Z 463.534,A -85,B 0,C 180,E1 -17678.423,E2 -17678.423} C_VEL
LIN {X 0,Y 285.845,Z 463.205,A -85,B 0,C 180,E1 -17680.342,E2 -17680.342} C_VEL
LIN {X 0,Y 284.915,Z 463.991,A -85,B 0,C 180,E1 -17682.267,E2 -17682.267} C_VEL
LIN {X 0,Y 284.349,Z 465.651,A -85,B 0,C 180,E1 -17684.211,E2 -17684.211} C_VEL
LIN {X 0,Y 284.137,Z 469.79,A -85,B 0,C 180,E1 -17686.937,E2 -17686.937} C_VEL
LIN {X 0,Y 284.618,Z 474.486,A -85,B 0,C 180,E1 -17689.213,E2 -17689.213} C_VEL
LIN {X 0,Y 285.12,Z 479.956,A -85,B 0,C 180,E1 -17691.092,E2 -17691.092} C_VEL
LIN {X 0,Y 285.098,Z 486.462,A -85,B 0,C 180,E1 -17692.654,E2 -17692.654} C_VEL
LIN {X 0,Y 285.285,Z 491.057,A -85,B 0,C 180,E1 -17693.754,E2 -17693.754} C_VEL
LIN {X 0,Y 285.616,Z 502.372,A -85,B 0,C 180,E1 -17696.212,E2 -17696.212} C_VEL
LIN {X 0,Y 285.395,Z 515.959,A -85,B 0,C 180,E1 -17698.859,E2 -17698.859} C_VEL
LIN {X 0,Y 284.549,Z 527.841,A -85,B 0,C 180,E1 -17701.088,E2 -17701.088} C_VEL
LIN {X 0,Y 283.224,Z 538.211,A -85,B 0,C 180,E1 -17703.072,E2 -17703.072} C_VEL
LIN {X 0,Y 280.189,Z 550.733,A -85,B 0,C 180,E1 -17705.551,E2 -17705.551} C_VEL
LIN {X 0,Y 277.337,Z 561.359,A -85,B 0,C 180,E1 -17708.051,E2 -17708.051} C_VEL
LIN {X 0,Y 274.201,Z 570.405,A -85,B 0,C 180,E1 -17710.536,E2 -17710.536} C_VEL
LIN {X 0,Y 271.455,Z 578.767,A -85,B 0,C 180,E1 -17713.453,E2 -17713.453} C_VEL
LIN {X 0,Y 270.156,Z 583.859,A -85,B 0,C 180,E1 -17715.691,E2 -17715.691} C_VEL
LIN {X 0,Y 269.185,Z 589.227,A -85,B 0,C 180,E1 -17718.707,E2 -17718.707} C_VEL
LIN {X 0,Y 269.037,Z 594.324,A -85,B 0,C 180,E1 -17721.739,E2 -17721.739} C_VEL
LIN {X 0,Y 269.229,Z 597.116,A -85,B 0,C 180,E1 -17724.006,E2 -17724.006} C_VEL
LIN {X 0,Y 269.513,Z 598.469,A -85,B 0,C 180,E1 -17725.513,E2 -17725.513} C_VEL
LIN {X 0,Y 270.129,Z 599.84,A -85,B 0,C 180,E1 -17728.509,E2 -17728.509} C_VEL
LIN {X 0,Y 270.516,Z 599.917,A -85,B 0,C 180,E1 -17730,E2 -17730} C_VEL
LIN {X 0,Y 270.135,Z 599.474,A -85,B 0,C 180,E1 -17731.49,E2 -17731.49} C_VEL
LIN {X 0,Y 269.793,Z 598.59,A -85,B 0,C 180,E1 -17732.986,E2 -17732.986} C_VEL
LIN {X 0,Y 269.62,Z 597.284,A -85,B 0,C 180,E1 -17734.485,E2 -17734.485} C_VEL
LIN {X 0,Y 269.238,Z 593.682,A -85,B 0,C 180,E1 -17737.285,E2 -17737.285} C_VEL
